LIN {X 0,Y 421.799,Z 977.518,A -85,B 0,C 180,E1 9515.942,E2 9515.942} C_VEL
LIN {X 0,Y 421.821,Z 978.492,A -85,B 0,C 180,E1 9519.003,E2 9519.003} C_VEL
LIN {X 0,Y 422.337,Z 975.375,A -85,B 0,C 180,E1 9522.556,E2 9522.556} C_VEL
LIN {X 0,Y 423.104,Z 967.595,A -85,B 0,C 180,E1 9526.055,E2 9526.055} C_VEL
LIN {X 0,Y 424.505,Z 953.17,A -85,B 0,C 180,E1 9529.758,E2 9529.758} C_VEL
LIN {X 0,Y 426.108,Z 934.517,A -85,B 0,C 180,E1 9532.847,E2 9532.847} C_VEL
LIN {X 0,Y 427.847,Z 910.65,A -85,B 0,C 180,E1 9535.461,E2 9535.461} C_VEL
LIN {X 0,Y 428.281,Z 890.231,A -85,B 0,C 180,E1 9537.014,E2 9537.014} C_VEL
LIN {X 0,Y 421.324,Z 861.271,A -85,B 0,C 180,E1 9538.781,E2 9538.781} C_VEL
LIN {X 0,Y 420.341,Z 857.28,A -85,B 0,C 180,E1 9538.956,E2 9538.956} C_VEL
LIN {X 0,Y 420.221,Z 857.28,A -85,B 0,C 180,E1 9544.157,E2 9544.157} C_VEL
LIN {X 0,Y 419.876,Z 857.28,A -85,B 0,C 180,E1 9550.41,E2 9550.41} C_VEL
LIN {X 0,Y 419.681,Z 857.28,A -85,B 0,C 180,E1 9556.795,E2 9556.795} C_VEL
LIN {X 0,Y 419.429,Z 857.28,A -85,B 0,C 180,E1 9563.414,E2 9563.414} C_VEL
LIN {X 0,Y 419.233,Z 857.28,A -85,B 0,C 180,E1 9570.388,E2 9570.388} C_VEL
LIN {X 0,Y 419.085,Z 857.28,A -85,B 0,C 180,E1 9577.363,E2 9577.363} C_VEL
LIN {X 0,Y 419.026,Z 857.28,A -85,B 0,C 180,E1 9583.726,E2 9583.726} C_VEL
LIN {X 0,Y 419.097,Z 857.28,A -85,B 0,C 180,E1 9589.438,E2 9589.438} C_VEL
LIN {X 0,Y 419.103,Z 857.28,A -85,B 0,C 180,E1 9596.203,E2 9596.203} C_VEL
LIN {X 0,Y 419.305,Z 857.723,A -85,B 0,C 180,E1 9598.793,E2 9598.793} C_VEL
LIN {X 0,Y 435.902,Z 903.66,A -85,B 0,C 180,E1 9600.619,E2 9600.619} C_VEL
LIN {X 0,Y 434.861,Z 940.44,A -85,B 0,C 180,E1 9601.516,E2 9601.516} C_VEL
LIN {X 0,Y 432.279,Z 973.093,A -85,B 0,C 180,E1 9603.034,E2 9603.034} C_VEL
LIN {X 0,Y 429.214,Z 1005.135,A -85,B 0,C 180,E1 9605.375,E2 9605.375} C_VEL
LIN {X 0,Y 428.851,Z 1008.694,A -85,B 0,C 180,E1 9605.694,E2 9605.694} C_VEL
LIN {X 0,Y 423.506,Z 1022.555,A -85,B 0,C 180,E1 9606.951,E2 9606.951} C_VEL
LIN {X 0,Y 418.257,Z 1035.44,A -85,B 0,C 180,E1 9608.402,E2 9608.402} C_VEL
LIN {X 0,Y 415.552,Z 1060.439,A -85,B 0,C 180,E1 9612.286,E2 9612.286} C_VEL
LIN {X 0,Y 414.019,Z 1079.134,A -85,B 0,C 180,E1 9616.393,E2 9616.393} C_VEL
LIN {X 0,Y 413.338,Z 1093.536,A -85,B 0,C 180,E1 9621.098,E2 9621.098} C_VEL
LIN {X 0,Y 413.202,Z 1101.646,A -85,B 0,C 180,E1 9625.798,E2 9625.798} C_VEL
LIN {X 0,Y 413.219,Z 1103.917,A -85,B 0,C 180,E1 9630.001,E2 9630.001} C_VEL
LIN {X 0,Y 413.204,Z 1101.557,A -85,B 0,C 180,E1 9634.203,E2 9634.203} C_VEL
LIN {X 0,Y 413.391,Z 1093.361,A -85,B 0,C 180,E1 9638.902,E2 9638.902} C_VEL
LIN {X 0,Y 414.016,Z 1078.868,A -85,B 0,C 180,E1 9643.605,E2 9643.605} C_VEL
LIN {X 0,Y 415.715,Z 1058.786,A -85,B 0,C 180,E1 9647.961,E2 9647.961} C_VEL
LIN {X 0,Y 418.387,Z 1034.343,A -85,B 0,C 180,E1 9651.712,E2 9651.712} C_VEL
LIN {X 0,Y 421.663,Z 1004.833,A -85,B 0,C 180,E1 9654.956,E2 9654.956} C_VEL
LIN {X 0,Y 425.056,Z 972.788,A -85,B 0,C 180,E1 9657.388,E2 9657.388} C_VEL
LIN {X 0,Y 427.787,Z 939.248,A -85,B 0,C 180,E1 9659.006,E2 9659.006} C_VEL
LIN {X 0,Y 428.561,Z 904.937,A -85,B 0,C 180,E1 9659.915,E2 9659.915} C_VEL
LIN {X 0,Y 412.812,Z 861.837,A -85,B 0,C 180,E1 9661.896,E2 9661.896} C_VEL
LIN {X 0,Y 411.31,Z 857.28,A -85,B 0,C 180,E1 9662.139,E2 9662.139} C_VEL
LIN {X 0,Y 411.036,Z 857.28,A -85,B 0,C 180,E1 9669.314,E2 9669.314} C_VEL
LIN {X 0,Y 411.046,Z 857.28,A -85,B 0,C 180,E1 9675.571,E2 9675.571} C_VEL
LIN {X 0,Y 411.109,Z 857.28,A -85,B 0,C 180,E1 9681.223,E2 9681.223} C_VEL
LIN {X 0,Y 411.195,Z 857.28,A -85,B 0,C 180,E1 9687.877,E2 9687.877} C_VEL
LIN {X 0,Y 411.371,Z 857.28,A -85,B 0,C 180,E1 9693.772,E2 9693.772} C_VEL
LIN {X 0,Y 411.659,Z 857.28,A -85,B 0,C 180,E1 9700.65,E2 9700.65} C_VEL
LIN {X 0,Y 411.735,Z 857.28,A -85,B 0,C 180,E1 9707.231,E2 9707.231} C_VEL
LIN {X 0,Y 412.172,Z 857.28,A -85,B 0,C 180,E1 9713.649,E2 9713.649} C_VEL
LIN {X 0,Y 412.461,Z 857.28,A -85,B 0,C 180,E1 9719.973,E2 9719.973} C_VEL
LIN {X 0,Y 412.137,Z 857.28,A -85,B 0,C 180,E1 9726.298,E2 9726.298} C_VEL
LIN {X 0,Y 411.881,Z 857.28,A -85,B 0,C 180,E1 9732.709,E2 9732.709} C_VEL
LIN {X 0,Y 411.647,Z 857.28,A -85,B 0,C 180,E1 9739.294,E2 9739.294} C_VEL
LIN {X 0,Y 411.376,Z 857.28,A -85,B 0,C 180,E1 9746.168,E2 9746.168} C_VEL
LIN {X 0,Y 411.191,Z 857.28,A -85,B 0,C 180,E1 9753.478,E2 9753.478} C_VEL
LIN {X 0,Y 411.021,Z 857.28,A -85,B 0,C 180,E1 9759.323,E2 9759.323} C_VEL
LIN {X 0,Y 411.073,Z 857.28,A -85,B 0,C 180,E1 9765.587,E2 9765.587} C_VEL
LIN {X 0,Y 411.258,Z 858.026,A -85,B 0,C 180,E1 9769.388,E2 9769.388} C_VEL
LIN {X 0,Y 420.757,Z 885.763,A -85,B 0,C 180,E1 9771.654,E2 9771.654} C_VEL
LIN {X 0,Y 423.982,Z 903.449,A -85,B 0,C 180,E1 9773.33,E2 9773.33} C_VEL
LIN {X 0,Y 421.34,Z 927.161,A -85,B 0,C 180,E1 9775.806,E2 9775.806} C_VEL
LIN {X 0,Y 418.651,Z 947.375,A -85,B 0,C 180,E1 9778.907,E2 9778.907} C_VEL
LIN {X 0,Y 416.418,Z 963.462,A -85,B 0,C 180,E1 9782.618,E2 9782.618} C_VEL
LIN {X 0,Y 415.038,Z 973.478,A -85,B 0,C 180,E1 9786.341,E2 9786.341} C_VEL
LIN {X 0,Y 414.274,Z 978.346,A -85,B 0,C 180,E1 9789.683,E2 9789.683} C_VEL
LIN {X 0,Y 413.931,Z 979.64,A -85,B 0,C 180,E1 9792.984,E2 9792.984} C_VEL
LIN {X 0,Y 414.318,Z 976.181,A -85,B 0,C 180,E1 9797.333,E2 9797.333} C_VEL
LIN {X 0,Y 415.259,Z 967.92,A -85,B 0,C 180,E1 9801.182,E2 9801.182} C_VEL
LIN {X 0,Y 416.858,Z 953.381,A -85,B 0,C 180,E1 9805.118,E2 9805.118} C_VEL
LIN {X 0,Y 419.039,Z 934.423,A -85,B 0,C 180,E1 9808.446,E2 9808.446} C_VEL
LIN {X 0,Y 421.351,Z 911.694,A -85,B 0,C 180,E1 9811.157,E2 9811.157} C_VEL
LIN {X 0,Y 422.02,Z 896.901,A -85,B 0,C 180,E1 9812.479,E2 9812.479} C_VEL
LIN {X 0,Y 415.522,Z 868.738,A -85,B 0,C 180,E1 9814.702,E2 9814.702} C_VEL
LIN {X 0,Y 412.172,Z 857.28,A -85,B 0,C 180,E1 9815.467,E2 9815.467} C_VEL
LIN {X 0,Y 411.961,Z 857.28,A -85,B 0,C 180,E1 9820.588,E2 9820.588} C_VEL
LIN {X 0,Y 411.718,Z 857.28,A -85,B 0,C 180,E1 9827.204,E2 9827.204} C_VEL
LIN {X 0,Y 411.416,Z 857.28,A -85,B 0,C 180,E1 9833.879,E2 9833.879} C_VEL
LIN {X 0,Y 411.283,Z 857.28,A -85,B 0,C 180,E1 9838.592,E2 9838.592} C_VEL
LIN {X 0,Y 411.132,Z 857.28,A -85,B 0,C 180,E1 9845.965,E2 9845.965} C_VEL
LIN {X 0,Y 411.032,Z 857.28,A -85,B 0,C 180,E1 9852.614,E2 9852.614} C_VEL
LIN {X 0,Y 411.302,Z 857.817,A -85,B 0,C 180,E1 9857,E2 9857} C_VEL
LIN {X 0,Y 418.345,Z 886.44,A -85,B 0,C 180,E1 9858.675,E2 9858.675} C_VEL
LIN {X 0,Y 419.854,Z 900.249,A -85,B 0,C 180,E1 9859.729,E2 9859.729} C_VEL
LIN {X 0,Y 418.125,Z 925.773,A -85,B 0,C 180,E1 9862.184,E2 9862.184} C_VEL
LIN {X 0,Y 416.519,Z 946.375,A -85,B 0,C 180,E1 9865.146,E2 9865.146} C_VEL
LIN {X 0,Y 415.31,Z 962.435,A -85,B 0,C 180,E1 9868.598,E2 9868.598} C_VEL
LIN {X 0,Y 414.455,Z 973.607,A -85,B 0,C 180,E1 9872.458,E2 9872.458} C_VEL
LIN {X 0,Y 413.982,Z 979.017,A -85,B 0,C 180,E1 9876.318,E2 9876.318} C_VEL
LIN {X 0,Y 413.979,Z 979.761,A -85,B 0,C 180,E1 9878.586,E2 9878.586} C_VEL
LIN {X 0,Y 414.406,Z 977.789,A -85,B 0,C 180,E1 9881.791,E2 9881.791} C_VEL
LIN {X 0,Y 415.312,Z 970.04,A -85,B 0,C 180,E1 9885.788,E2 9885.788} C_VEL
LIN {X 0,Y 416.722,Z 956.488,A -85,B 0,C 180,E1 9889.565,E2 9889.565} C_VEL
LIN {X 0,Y 418.38,Z 938.471,A -85,B 0,C 180,E1 9892.753,E2 9892.753} C_VEL
LIN {X 0,Y 420.149,Z 916.25,A -85,B 0,C 180,E1 9895.392,E2 9895.392} C_VEL
LIN {X 0,Y 420.82,Z 891.257,A -85,B 0,C 180,E1 9897.396,E2 9897.396} C_VEL
LIN {X 0,Y 413.932,Z 863.039,A -85,B 0,C 180,E1 9899.176,E2 9899.176} C_VEL
LIN {X 0,Y 412.429,Z 857.28,A -85,B 0,C 180,E1 9899.501,E2 9899.501} C_VEL
LIN {X 0,Y 412.121,Z 857.28,A -85,B 0,C 180,E1 9906.352,E2 9906.352} C_VEL
LIN {X 0,Y 411.856,Z 857.28,A -85,B 0,C 180,E1 9912.765,E2 9912.765} C_VEL
LIN {X 0,Y 411.654,Z 857.28,A -85,B 0,C 180,E1 9919.351,E2 9919.351} C_VEL
LIN {X 0,Y 411.368,Z 857.28,A -85,B 0,C 180,E1 9926.228,E2 9926.228} C_VEL
LIN {X 0,Y 411.217,Z 857.28,A -85,B 0,C 180,E1 9933.54,E2 9933.54} C_VEL
LIN {X 0,Y 411.052,Z 857.28,A -85,B 0,C 180,E1 9939.33,E2 9939.33} C_VEL
LIN {X 0,Y 411.092,Z 857.28,A -85,B 0,C 180,E1 9945.592,E2 9945.592} C_VEL
LIN {X 0,Y 411.112,Z 857.28,A -85,B 0,C 180,E1 9951.239,E2 9951.239} C_VEL
LIN {X 0,Y 411.368,Z 857.28,A -85,B 0,C 180,E1 9958.268,E2 9958.268} C_VEL
LIN {X 0,Y 428.788,Z 907.527,A -85,B 0,C 180,E1 9960.271,E2 9960.271} C_VEL
LIN {X 0,Y 427.327,Z 943.567,A -85,B 0,C 180,E1 9961.236,E2 9961.236} C_VEL
LIN {X 0,Y 424.531,Z 976.772,A -85,B 0,C 180,E1 9962.901,E2 9962.901} C_VEL
LIN {X 0,Y 421.193,Z 1009.104,A -85,B 0,C 180,E1 9965.441,E2 9965.441} C_VEL
LIN {X 0,Y 418.257,Z 1035.44,A -85,B 0,C 180,E1 9968.402,E2 9968.402} C_VEL
LIN {X 0,Y 416.387,Z 1041.625,A -85,B 0,C 180,E1 9969.217,E2 9969.217} C_VEL
LIN {X 0,Y 408.17,Z 1056.964,A -85,B 0,C 180,E1 9971.556,E2 9971.556} C_VEL
LIN {X 0,Y 407.937,Z 1058.282,A -85,B 0,C 180,E1 9971.801,E2 9971.801} C_VEL
LIN {X 0,Y 406.3,Z 1076.772,A -85,B 0,C 180,E1 9975.845,E2 9975.845} C_VEL
LIN {X 0,Y 405.5,Z 1090.903,A -85,B 0,C 180,E1 9980.328,E2 9980.328} C_VEL
LIN {X 0,Y 405.399,Z 1099.167,A -85,B 0,C 180,E1 9984.643,E2 9984.643} C_VEL
LIN {X 0,Y 405.33,Z 1102.132,A -85,B 0,C 180,E1 9987.86,E2 9987.86} C_VEL
LIN {X 0,Y 405.334,Z 1102.085,A -85,B 0,C 180,E1 9992.141,E2 9992.141} C_VEL
LIN {X 0,Y 405.37,Z 1097.398,A -85,B 0,C 180,E1 9996.434,E2 9996.434} C_VEL
LIN {X 0,Y 405.594,Z 1087.82,A -85,B 0,C 180,E1 10000.758,E2 10000.758} C_VEL
LIN {X 0,Y 406.651,Z 1071.54,A -85,B 0,C 180,E1 10005.385,E2 10005.385} C_VEL
LIN {X 0,Y 408.664,Z 1050.837,A -85,B 0,C 180,E1 10009.479,E2 10009.479} C_VEL
LIN {X 0,Y 411.694,Z 1025.006,A -85,B 0,C 180,E1 10013.148,E2 10013.148} C_VEL
LIN {X 0,Y 415.216,Z 995.793,A -85,B 0,C 180,E1 10016.108,E2 10016.108} C_VEL
LIN {X 0,Y 418.709,Z 963.598,A -85,B 0,C 180,E1 10018.343,E2 10018.343} C_VEL
LIN {X 0,Y 421.277,Z 930.208,A -85,B 0,C 180,E1 10019.771,E2 10019.771} C_VEL
LIN {X 0,Y 421.345,Z 906.279,A -85,B 0,C 180,E1 10020.4,E2 10020.4} C_VEL
LIN {X 0,Y 407.006,Z 866.784,A -85,B 0,C 180,E1 10022.269,E2 10022.269} C_VEL
LIN {X 0,Y 403.353,Z 857.28,A -85,B 0,C 180,E1 10022.88,E2 10022.88} C_VEL
LIN {X 0,Y 403.089,Z 857.28,A -85,B 0,C 180,E1 10029.685,E2 10029.685} C_VEL
LIN {X 0,Y 403.143,Z 857.28,A -85,B 0,C 180,E1 10035.528,E2 10035.528} C_VEL
LIN {X 0,Y 403.133,Z 857.28,A -85,B 0,C 180,E1 10042.067,E2 10042.067} C_VEL
LIN {X 0,Y 403.303,Z 857.28,A -85,B 0,C 180,E1 10048.275,E2 10048.275} C_VEL
LIN {X 0,Y 403.503,Z 857.28,A -85,B 0,C 180,E1 10055.603,E2 10055.603} C_VEL
LIN {X 0,Y 403.726,Z 857.28,A -85,B 0,C 180,E1 10062.52,E2 10062.52} C_VEL
LIN {X 0,Y 403.89,Z 857.28,A -85,B 0,C 180,E1 10069.174,E2 10069.174} C_VEL
LIN {X 0,Y 404.284,Z 857.28,A -85,B 0,C 180,E1 10075.679,E2 10075.679} C_VEL
LIN {X 0,Y 404.458,Z 857.28,A -85,B 0,C 180,E1 10082.117,E2 10082.117} C_VEL
LIN {X 0,Y 404.116,Z 857.28,A -85,B 0,C 180,E1 10088.588,E2 10088.588} C_VEL
LIN {X 0,Y 403.867,Z 857.28,A -85,B 0,C 180,E1 10095.179,E2 10095.179} C_VEL
LIN {X 0,Y 403.608,Z 857.28,A -85,B 0,C 180,E1 10101.993,E2 10101.993} C_VEL
LIN {X 0,Y 403.322,Z 857.28,A -85,B 0,C 180,E1 10109.165,E2 10109.165} C_VEL
LIN {X 0,Y 403.218,Z 857.28,A -85,B 0,C 180,E1 10114.299,E2 10114.299} C_VEL
LIN {X 0,Y 403.087,Z 857.28,A -85,B 0,C 180,E1 10121.301,E2 10121.301} C_VEL
LIN {X 0,Y 403.18,Z 857.28,A -85,B 0,C 180,E1 10127.47,E2 10127.47} C_VEL
LIN {X 0,Y 403.25,Z 857.838,A -85,B 0,C 180,E1 10128.673,E2 10128.673} C_VEL
LIN {X 0,Y 412.99,Z 885.391,A -85,B 0,C 180,E1 10130.993,E2 10130.993} C_VEL
LIN {X 0,Y 416.797,Z 905.603,A -85,B 0,C 180,E1 10132.975,E2 10132.975} C_VEL
LIN {X 0,Y 413.764,Z 930.558,A -85,B 0,C 180,E1 10135.701,E2 10135.701} C_VEL
LIN {X 0,Y 410.953,Z 950.524,A -85,B 0,C 180,E1 10138.948,E2 10138.948} C_VEL
LIN {X 0,Y 408.665,Z 965.697,A -85,B 0,C 180,E1 10142.663,E2 10142.663} C_VEL
LIN {X 0,Y 407.065,Z 976.221,A -85,B 0,C 180,E1 10147.011,E2 10147.011} C_VEL
LIN {X 0,Y 406.352,Z 980.147,A -85,B 0,C 180,E1 10150.406,E2 10150.406} C_VEL
LIN {X 0,Y 406.187,Z 980.065,A -85,B 0,C 180,E1 10154.874,E2 10154.874} C_VEL
LIN {X 0,Y 406.935,Z 974.024,A -85,B 0,C 180,E1 10159.278,E2 10159.278} C_VEL
LIN {X 0,Y 408.182,Z 963.556,A -85,B 0,C 180,E1 10163.075,E2 10163.075} C_VEL
LIN {X 0,Y 410.029,Z 946.849,A -85,B 0,C 180,E1 10166.87,E2 10166.87} C_VEL
LIN {X 0,Y 412.625,Z 925.085,A -85,B 0,C 180,E1 10170.131,E2 10170.131} C_VEL
LIN {X 0,Y 414.937,Z 900.466,A -85,B 0,C 180,E1 10172.614,E2 10172.614} C_VEL
LIN {X 0,Y 408.725,Z 872.434,A -85,B 0,C 180,E1 10174.946,E2 10174.946} C_VEL
LIN {X 0,Y 404.281,Z 857.28,A -85,B 0,C 180,E1 10176.045,E2 10176.045} C_VEL
LIN {X 0,Y 403.946,Z 857.28,A -85,B 0,C 180,E1 10183.186,E2 10183.186} C_VEL
LIN {X 0,Y 403.666,Z 857.28,A -85,B 0,C 180,E1 10189.728,E2 10189.728} C_VEL
LIN {X 0,Y 403.392,Z 857.28,A -85,B 0,C 180,E1 10196.769,E2 10196.769} C_VEL
LIN {X 0,Y 403.237,Z 857.28,A -85,B 0,C 180,E1 10201.713,E2 10201.713} C_VEL
LIN {X 0,Y 403.069,Z 857.28,A -85,B 0,C 180,E1 10208,E2 10208} C_VEL
LIN {X 0,Y 403.179,Z 857.28,A -85,B 0,C 180,E1 10214.543,E2 10214.543} C_VEL
LIN {X 0,Y 403.347,Z 857.28,A -85,B 0,C 180,E1 10216.554,E2 10216.554} C_VEL
LIN {X 0,Y 410.553,Z 886.738,A -85,B 0,C 180,E1 10218.313,E2 10218.313} C_VEL
LIN {X 0,Y 412.256,Z 902.112,A -85,B 0,C 180,E1 10219.511,E2 10219.511} C_VEL
LIN {X 0,Y 410.519,Z 926.722,A -85,B 0,C 180,E1 10221.928,E2 10221.928} C_VEL
LIN {X 0,Y 408.827,Z 947.408,A -85,B 0,C 180,E1 10224.943,E2 10224.943} C_VEL
LIN {X 0,Y 407.561,Z 963.335,A -85,B 0,C 180,E1 10228.403,E2 10228.403} C_VEL
LIN {X 0,Y 406.687,Z 974.589,A -85,B 0,C 180,E1 10232.311,E2 10232.311} C_VEL
LIN {X 0,Y 406.202,Z 979.817,A -85,B 0,C 180,E1 10235.835,E2 10235.835} C_VEL
LIN {X 0,Y 406.194,Z 980.973,A -85,B 0,C 180,E1 10238.726,E2 10238.726} C_VEL
LIN {X 0,Y 406.813,Z 977.958,A -85,B 0,C 180,E1 10242.714,E2 10242.714} C_VEL
LIN {X 0,Y 407.768,Z 969.392,A -85,B 0,C 180,E1 10246.652,E2 10246.652} C_VEL
LIN {X 0,Y 409.425,Z 954.746,A -85,B 0,C 180,E1 10250.452,E2 10250.452} C_VEL
LIN {X 0,Y 411.31,Z 935.202,A -85,B 0,C 180,E1 10253.69,E2 10253.69} C_VEL
LIN {X 0,Y 413.177,Z 912.352,A -85,B 0,C 180,E1 10256.22,E2 10256.22} C_VEL
LIN {X 0,Y 413.681,Z 893.995,A -85,B 0,C 180,E1 10257.668,E2 10257.668} C_VEL
LIN {X 0,Y 407.079,Z 866.072,A -85,B 0,C 180,E1 10259.518,E2 10259.518} C_VEL
LIN {X 0,Y 404.546,Z 857.28,A -85,B 0,C 180,E1 10260.027,E2 10260.027} C_VEL
LIN {X 0,Y 404.205,Z 857.28,A -85,B 0,C 180,E1 10266.477,E2 10266.477} C_VEL
LIN {X 0,Y 403.943,Z 857.28,A -85,B 0,C 180,E1 10273.019,E2 10273.019} C_VEL
LIN {X 0,Y 403.691,Z 857.28,A -85,B 0,C 180,E1 10279.748,E2 10279.748} C_VEL
LIN {X 0,Y 403.436,Z 857.28,A -85,B 0,C 180,E1 10286.785,E2 10286.785} C_VEL
LIN {X 0,Y 403.305,Z 857.28,A -85,B 0,C 180,E1 10291.725,E2 10291.725} C_VEL
LIN {X 0,Y 403.088,Z 857.28,A -85,B 0,C 180,E1 10297.928,E2 10297.928} C_VEL
LIN {X 0,Y 403.176,Z 857.28,A -85,B 0,C 180,E1 10304.479,E2 10304.479} C_VEL
LIN {X 0,Y 403.172,Z 857.28,A -85,B 0,C 180,E1 10310.327,E2 10310.327} C_VEL
LIN {X 0,Y 403.41,Z 857.488,A -85,B 0,C 180,E1 10317.744,E2 10317.744} C_VEL
LIN {X 0,Y 421.549,Z 909.75,A -85,B 0,C 180,E1 10319.877,E2 10319.877} C_VEL
LIN {X 0,Y 419.914,Z 945.02,A -85,B 0,C 180,E1 10320.888,E2 10320.888} C_VEL
LIN {X 0,Y 416.875,Z 978.864,A -85,B 0,C 180,E1 10322.687,E2 10322.687} C_VEL
LIN {X 0,Y 413.474,Z 1009.986,A -85,B 0,C 180,E1 10325.24,E2 10325.24} C_VEL
LIN {X 0,Y 410.12,Z 1038.585,A -85,B 0,C 180,E1 10328.62,E2 10328.62} C_VEL
LIN {X 0,Y 407.937,Z 1058.282,A -85,B 0,C 180,E1 10331.801,E2 10331.801} C_VEL
LIN {X 0,Y 403.019,Z 1068.016,A -85,B 0,C 180,E1 10333.752,E2 10333.752} C_VEL
LIN {X 0,Y 398.406,Z 1076.498,A -85,B 0,C 180,E1 10335.847,E2 10335.847} C_VEL
LIN {X 0,Y 397.627,Z 1090.953,A -85,B 0,C 180,E1 10340.688,E2 10340.688} C_VEL
LIN {X 0,Y 397.57,Z 1097.979,A -85,B 0,C 180,E1 10344.537,E2 10344.537} C_VEL
LIN {X 0,Y 397.506,Z 1100.956,A -85,B 0,C 180,E1 10347.818,E2 10347.818} C_VEL
LIN {X 0,Y 397.51,Z 1100.908,A -85,B 0,C 180,E1 10352.184,E2 10352.184} C_VEL
LIN {X 0,Y 397.55,Z 1096.206,A -85,B 0,C 180,E1 10356.561,E2 10356.561} C_VEL
LIN {X 0,Y 397.751,Z 1086.607,A -85,B 0,C 180,E1 10360.973,E2 10360.973} C_VEL
LIN {X 0,Y 398.894,Z 1070.287,A -85,B 0,C 180,E1 10365.691,E2 10365.691} C_VEL
LIN {X 0,Y 401.197,Z 1047.885,A -85,B 0,C 180,E1 10370.144,E2 10370.144} C_VEL
LIN {X 0,Y 404.421,Z 1022.323,A -85,B 0,C 180,E1 10373.772,E2 10373.772} C_VEL
LIN {X 0,Y 408.187,Z 992.517,A -85,B 0,C 180,E1 10376.773,E2 10376.773} C_VEL
LIN {X 0,Y 411.785,Z 960.401,A -85,B 0,C 180,E1 10378.967,E2 10378.967} C_VEL
LIN {X 0,Y 414.481,Z 926.066,A -85,B 0,C 180,E1 10380.394,E2 10380.394} C_VEL
LIN {X 0,Y 414.518,Z 908.545,A -85,B 0,C 180,E1 10380.854,E2 10380.854} C_VEL
LIN {X 0,Y 400.695,Z 870.24,A -85,B 0,C 180,E1 10382.732,E2 10382.732} C_VEL
LIN {X 0,Y 395.38,Z 857.28,A -85,B 0,C 180,E1 10383.539,E2 10383.539} C_VEL
LIN {X 0,Y 395.178,Z 857.28,A -85,B 0,C 180,E1 10390.643,E2 10390.643} C_VEL
LIN {X 0,Y 395.204,Z 857.28,A -85,B 0,C 180,E1 10396.713,E2 10396.713} C_VEL
LIN {X 0,Y 395.224,Z 857.28,A -85,B 0,C 180,E1 10403.563,E2 10403.563} C_VEL
LIN {X 0,Y 395.422,Z 857.28,A -85,B 0,C 180,E1 10410.129,E2 10410.129} C_VEL
LIN {X 0,Y 395.654,Z 857.28,A -85,B 0,C 180,E1 10417.48,E2 10417.48} C_VEL
LIN {X 0,Y 395.796,Z 857.28,A -85,B 0,C 180,E1 10424.446,E2 10424.446} C_VEL
LIN {X 0,Y 396.18,Z 857.28,A -85,B 0,C 180,E1 10431.182,E2 10431.182} C_VEL
LIN {X 0,Y 396.624,Z 857.28,A -85,B 0,C 180,E1 10437.785,E2 10437.785} C_VEL
LIN {X 0,Y 396.46,Z 857.28,A -85,B 0,C 180,E1 10444.351,E2 10444.351} C_VEL
LIN {X 0,Y 396.105,Z 857.28,A -85,B 0,C 180,E1 10450.985,E2 10450.985} C_VEL
LIN {X 0,Y 395.861,Z 857.28,A -85,B 0,C 180,E1 10457.78,E2 10457.78} C_VEL
LIN {X 0,Y 395.562,Z 857.28,A -85,B 0,C 180,E1 10464.858,E2 10464.858} C_VEL
LIN {X 0,Y 395.39,Z 857.28,A -85,B 0,C 180,E1 10469.809,E2 10469.809} C_VEL
LIN {X 0,Y 395.164,Z 857.28,A -85,B 0,C 180,E1 10476.425,E2 10476.425} C_VEL
LIN {X 0,Y 395.176,Z 857.28,A -85,B 0,C 180,E1 10483.54,E2 10483.54} C_VEL
LIN {X 0,Y 395.303,Z 857.752,A -85,B 0,C 180,E1 10487.932,E2 10487.932} C_VEL
LIN {X 0,Y 405.656,Z 886.594,A -85,B 0,C 180,E1 10490.452,E2 10490.452} C_VEL
LIN {X 0,Y 409.752,Z 906.655,A -85,B 0,C 180,E1 10492.504,E2 10492.504} C_VEL
LIN {X 0,Y 406.609,Z 931.138,A -85,B 0,C 180,E1 10495.212,E2 10495.212} C_VEL
LIN {X 0,Y 403.574,Z 951.34,A -85,B 0,C 180,E1 10498.533,E2 10498.533} C_VEL
LIN {X 0,Y 400.976,Z 967.421,A -85,B 0,C 180,E1 10502.576,E2 10502.576} C_VEL
LIN {X 0,Y 399.409,Z 976.939,A -85,B 0,C 180,E1 10506.544,E2 10506.544} C_VEL
LIN {X 0,Y 398.598,Z 981.128,A -85,B 0,C 180,E1 10510.009,E2 10510.009} C_VEL
LIN {X 0,Y 398.358,Z 981.404,A -85,B 0,C 180,E1 10514.569,E2 10514.569} C_VEL
LIN {X 0,Y 399.089,Z 975.816,A -85,B 0,C 180,E1 10519.064,E2 10519.064} C_VEL
LIN {X 0,Y 400.311,Z 965.763,A -85,B 0,C 180,E1 10522.938,E2 10522.938} C_VEL
LIN {X 0,Y 402.252,Z 949.494,A -85,B 0,C 180,E1 10526.832,E2 10526.832} C_VEL
LIN {X 0,Y 404.884,Z 928.588,A -85,B 0,C 180,E1 10530.133,E2 10530.133} C_VEL
LIN {X 0,Y 407.504,Z 903.528,A -85,B 0,C 180,E1 10532.801,E2 10532.801} C_VEL
LIN {X 0,Y 402.018,Z 876.594,A -85,B 0,C 180,E1 10535.158,E2 10535.158} C_VEL
LIN {X 0,Y 396.318,Z 857.28,A -85,B 0,C 180,E1 10536.58,E2 10536.58} C_VEL
LIN {X 0,Y 396.051,Z 857.28,A -85,B 0,C 180,E1 10543.26,E2 10543.26} C_VEL
LIN {X 0,Y 395.729,Z 857.28,A -85,B 0,C 180,E1 10550.141,E2 10550.141} C_VEL
LIN {X 0,Y 395.4,Z 857.28,A -85,B 0,C 180,E1 10557.355,E2 10557.355} C_VEL
LIN {X 0,Y 395.235,Z 857.28,A -85,B 0,C 180,E1 10562.656,E2 10562.656} C_VEL
LIN {X 0,Y 395.162,Z 857.28,A -85,B 0,C 180,E1 10570.05,E2 10570.05} C_VEL
LIN {X 0,Y 395.421,Z 857.731,A -85,B 0,C 180,E1 10576.204,E2 10576.204} C_VEL
LIN {X 0,Y 402.625,Z 886.578,A -85,B 0,C 180,E1 10577.908,E2 10577.908} C_VEL
LIN {X 0,Y 404.763,Z 902.529,A -85,B 0,C 180,E1 10579.168,E2 10579.168} C_VEL
LIN {X 0,Y 402.857,Z 928.419,A -85,B 0,C 180,E1 10581.752,E2 10581.752} C_VEL
LIN {X 0,Y 401.051,Z 949.418,A -85,B 0,C 180,E1 10584.913,E2 10584.913} C_VEL
LIN {X 0,Y 399.733,Z 966.013,A -85,B 0,C 180,E1 10588.695,E2 10588.695} C_VEL
LIN {X 0,Y 398.864,Z 976.061,A -85,B 0,C 180,E1 10592.39,E2 10592.39} C_VEL
LIN {X 0,Y 398.408,Z 980.97,A -85,B 0,C 180,E1 10595.792,E2 10595.792} C_VEL
LIN {X 0,Y 398.56,Z 981.853,A -85,B 0,C 180,E1 10600.046,E2 10600.046} C_VEL
LIN {X 0,Y 399.323,Z 977.179,A -85,B 0,C 180,E1 10604.08,E2 10604.08} C_VEL
LIN {X 0,Y 400.609,Z 966.545,A -85,B 0,C 180,E1 10608.147,E2 10608.147} C_VEL
LIN {X 0,Y 402.291,Z 951.37,A -85,B 0,C 180,E1 10611.646,E2 10611.646} C_VEL
LIN {X 0,Y 404.458,Z 930.239,A -85,B 0,C 180,E1 10614.829,E2 10614.829} C_VEL
LIN {X 0,Y 406.406,Z 906.173,A -85,B 0,C 180,E1 10617.226,E2 10617.226} C_VEL
LIN {X 0,Y 405.655,Z 891.937,A -85,B 0,C 180,E1 10618.333,E2 10618.333} C_VEL
LIN {X 0,Y 398.867,Z 864.613,A -85,B 0,C 180,E1 10620.13,E2 10620.13} C_VEL
LIN {X 0,Y 396.573,Z 857.28,A -85,B 0,C 180,E1 10620.575,E2 10620.575} C_VEL
LIN {X 0,Y 396.287,Z 857.28,A -85,B 0,C 180,E1 10626.607,E2 10626.607} C_VEL
LIN {X 0,Y 395.999,Z 857.28,A -85,B 0,C 180,E1 10633.285,E2 10633.285} C_VEL
LIN {X 0,Y 395.774,Z 857.28,A -85,B 0,C 180,E1 10640.16,E2 10640.16} C_VEL
LIN {X 0,Y 395.448,Z 857.28,A -85,B 0,C 180,E1 10647.37,E2 10647.37} C_VEL
LIN {X 0,Y 395.326,Z 857.28,A -85,B 0,C 180,E1 10652.587,E2 10652.587} C_VEL
LIN {X 0,Y 395.213,Z 857.28,A -85,B 0,C 180,E1 10659.987,E2 10659.987} C_VEL
LIN {X 0,Y 395.24,Z 857.28,A -85,B 0,C 180,E1 10666.721,E2 10666.721} C_VEL
LIN {X 0,Y 395.23,Z 857.28,A -85,B 0,C 180,E1 10673.574,E2 10673.574} C_VEL
LIN {X 0,Y 395.451,Z 857.28,A -85,B 0,C 180,E1 10677.177,E2 10677.177} C_VEL
LIN {X 0,Y 414.296,Z 909.828,A -85,B 0,C 180,E1 10679.434,E2 10679.434} C_VEL
LIN {X 0,Y 412.562,Z 945.735,A -85,B 0,C 180,E1 10680.501,E2 10680.501} C_VEL
LIN {X 0,Y 409.54,Z 977.826,A -85,B 0,C 180,E1 10682.251,E2 10682.251} C_VEL
LIN {X 0,Y 405.943,Z 1009.456,A -85,B 0,C 180,E1 10684.897,E2 10684.897} C_VEL
LIN {X 0,Y 402.556,Z 1036.966,A -85,B 0,C 180,E1 10688.198,E2 10688.198} C_VEL
LIN {X 0,Y 399.912,Z 1059.738,A -85,B 0,C 180,E1 10692.003,E2 10692.003} C_VEL
LIN {X 0,Y 398.406,Z 1076.498,A -85,B 0,C 180,E1 10695.847,E2 10695.847} C_VEL
LIN {X 0,Y 395.545,Z 1082.115,A -85,B 0,C 180,E1 10697.513,E2 10697.513} C_VEL
LIN {X 0,Y 389.884,Z 1088.855,A -85,B 0,C 180,E1 10700.117,E2 10700.117} C_VEL
LIN {X 0,Y 389.777,Z 1089.526,A -85,B 0,C 180,E1 10700.423,E2 10700.423} C_VEL
LIN {X 0,Y 389.742,Z 1096.776,A -85,B 0,C 180,E1 10704.427,E2 10704.427} C_VEL
LIN {X 0,Y 389.696,Z 1099.774,A -85,B 0,C 180,E1 10707.774,E2 10707.774} C_VEL
LIN {X 0,Y 389.7,Z 1099.736,A -85,B 0,C 180,E1 10712.227,E2 10712.227} C_VEL
LIN {X 0,Y 389.716,Z 1095.022,A -85,B 0,C 180,E1 10716.694,E2 10716.694} C_VEL
LIN {X 0,Y 389.908,Z 1085.395,A -85,B 0,C 180,E1 10721.196,E2 10721.196} C_VEL
LIN {X 0,Y 391.134,Z 1069.07,A -85,B 0,C 180,E1 10726.011,E2 10726.011} C_VEL
LIN {X 0,Y 393.354,Z 1048.307,A -85,B 0,C 180,E1 10730.27,E2 10730.27} C_VEL
LIN {X 0,Y 396.754,Z 1022.833,A -85,B 0,C 180,E1 10734.023,E2 10734.023} C_VEL
LIN {X 0,Y 400.75,Z 992.969,A -85,B 0,C 180,E1 10737.142,E2 10737.142} C_VEL
LIN {X 0,Y 404.541,Z 961.247,A -85,B 0,C 180,E1 10739.396,E2 10739.396} C_VEL
LIN {X 0,Y 407.347,Z 928.595,A -85,B 0,C 180,E1 10740.825,E2 10740.825} C_VEL
LIN {X 0,Y 407.443,Z 910.061,A -85,B 0,C 180,E1 10741.366,E2 10741.366} C_VEL
LIN {X 0,Y 394.116,Z 873.196,A -85,B 0,C 180,E1 10743.253,E2 10743.253} C_VEL
LIN {X 0,Y 387.397,Z 857.28,A -85,B 0,C 180,E1 10744.248,E2 10744.248} C_VEL
LIN {X 0,Y 387.178,Z 857.28,A -85,B 0,C 180,E1 10751.668,E2 10751.668} C_VEL
LIN {X 0,Y 387.228,Z 857.28,A -85,B 0,C 180,E1 10758.324,E2 10758.324} C_VEL
LIN {X 0,Y 387.359,Z 857.28,A -85,B 0,C 180,E1 10765.169,E2 10765.169} C_VEL
LIN {X 0,Y 387.541,Z 857.28,A -85,B 0,C 180,E1 10772.023,E2 10772.023} C_VEL
LIN {X 0,Y 387.835,Z 857.28,A -85,B 0,C 180,E1 10779.546,E2 10779.546} C_VEL
LIN {X 0,Y 387.914,Z 857.28,A -85,B 0,C 180,E1 10786.433,E2 10786.433} C_VEL
LIN {X 0,Y 388.451,Z 857.28,A -85,B 0,C 180,E1 10793.259,E2 10793.259} C_VEL
LIN {X 0,Y 388.763,Z 857.28,A -85,B 0,C 180,E1 10799.971,E2 10799.971} C_VEL
LIN {X 0,Y 388.404,Z 857.28,A -85,B 0,C 180,E1 10806.684,E2 10806.684} C_VEL
LIN {X 0,Y 388.072,Z 857.28,A -85,B 0,C 180,E1 10813.503,E2 10813.503} C_VEL
LIN {X 0,Y 387.797,Z 857.28,A -85,B 0,C 180,E1 10820.532,E2 10820.532} C_VEL
LIN {X 0,Y 387.523,Z 857.28,A -85,B 0,C 180,E1 10827.914,E2 10827.914} C_VEL
LIN {X 0,Y 387.275,Z 857.28,A -85,B 0,C 180,E1 10835.851,E2 10835.851} C_VEL
LIN {X 0,Y 387.154,Z 857.28,A -85,B 0,C 180,E1 10842.007,E2 10842.007} C_VEL
LIN {X 0,Y 387.348,Z 857.28,A -85,B 0,C 180,E1 10847.133,E2 10847.133} C_VEL
LIN {X 0,Y 398.064,Z 886.834,A -85,B 0,C 180,E1 10849.786,E2 10849.786} C_VEL
LIN {X 0,Y 402.64,Z 908.425,A -85,B 0,C 180,E1 10852.079,E2 10852.079} C_VEL
LIN {X 0,Y 399.36,Z 932.498,A -85,B 0,C 180,E1 10854.81,E2 10854.81} C_VEL
LIN {X 0,Y 396.245,Z 951.943,A -85,B 0,C 180,E1 10858.055,E2 10858.055} C_VEL
LIN {X 0,Y 393.647,Z 966.945,A -85,B 0,C 180,E1 10861.767,E2 10861.767} C_VEL
LIN {X 0,Y 391.781,Z 977.624,A -85,B 0,C 180,E1 10866.059,E2 10866.059} C_VEL
LIN {X 0,Y 390.883,Z 982.112,A -85,B 0,C 180,E1 10869.597,E2 10869.597} C_VEL
LIN {X 0,Y 390.517,Z 982.738,A -85,B 0,C 180,E1 10874.252,E2 10874.252} C_VEL
LIN {X 0,Y 391.21,Z 977.525,A -85,B 0,C 180,E1 10878.841,E2 10878.841} C_VEL
LIN {X 0,Y 392.46,Z 967.87,A -85,B 0,C 180,E1 10882.796,E2 10882.796} C_VEL
LIN {X 0,Y 394.399,Z 952.815,A -85,B 0,C 180,E1 10886.636,E2 10886.636} C_VEL
LIN {X 0,Y 396.975,Z 933.05,A -85,B 0,C 180,E1 10889.999,E2 10889.999} C_VEL
LIN {X 0,Y 399.784,Z 908.244,A -85,B 0,C 180,E1 10892.848,E2 10892.848} C_VEL
LIN {X 0,Y 398.444,Z 895.498,A -85,B 0,C 180,E1 10894.085,E2 10894.085} C_VEL
LIN {X 0,Y 391.725,Z 868.476,A -85,B 0,C 180,E1 10896.291,E2 10896.291} C_VEL
LIN {X 0,Y 388.372,Z 857.28,A -85,B 0,C 180,E1 10897.059,E2 10897.059} C_VEL
LIN {X 0,Y 388.116,Z 857.28,A -85,B 0,C 180,E1 10903.536,E2 10903.536} C_VEL
LIN {X 0,Y 387.758,Z 857.28,A -85,B 0,C 180,E1 10910.574,E2 10910.574} C_VEL
LIN {X 0,Y 387.463,Z 857.28,A -85,B 0,C 180,E1 10917.963,E2 10917.963} C_VEL
LIN {X 0,Y 387.268,Z 857.28,A -85,B 0,C 180,E1 10925.904,E2 10925.904} C_VEL
LIN {X 0,Y 387.175,Z 857.28,A -85,B 0,C 180,E1 10932.082,E2 10932.082} C_VEL
LIN {X 0,Y 387.446,Z 857.28,A -85,B 0,C 180,E1 10935.759,E2 10935.759} C_VEL
LIN {X 0,Y 394.762,Z 886.609,A -85,B 0,C 180,E1 10937.508,E2 10937.508} C_VEL
LIN {X 0,Y 397.189,Z 904.358,A -85,B 0,C 180,E1 10938.941,E2 10938.941} C_VEL
LIN {X 0,Y 395.259,Z 929.232,A -85,B 0,C 180,E1 10941.473,E2 10941.473} C_VEL
LIN {X 0,Y 393.347,Z 950.858,A -85,B 0,C 180,E1 10944.785,E2 10944.785} C_VEL
LIN {X 0,Y 391.954,Z 967.218,A -85,B 0,C 180,E1 10948.591,E2 10948.591} C_VEL
LIN {X 0,Y 391.069,Z 977.282,A -85,B 0,C 180,E1 10952.361,E2 10952.361} C_VEL
LIN {X 0,Y 390.683,Z 981.15,A -85,B 0,C 180,E1 10954.81,E2 10954.81} C_VEL
LIN {X 0,Y 390.601,Z 983.414,A -85,B 0,C 180,E1 10958.48,E2 10958.48} C_VEL
LIN {X 0,Y 391.343,Z 980.175,A -85,B 0,C 180,E1 10963.169,E2 10963.169} C_VEL
LIN {X 0,Y 392.504,Z 971.47,A -85,B 0,C 180,E1 10967.22,E2 10967.22} C_VEL
LIN {X 0,Y 394.265,Z 957.644,A -85,B 0,C 180,E1 10970.932,E2 10970.932} C_VEL
LIN {X 0,Y 396.395,Z 938.521,A -85,B 0,C 180,E1 10974.253,E2 10974.253} C_VEL
LIN {X 0,Y 398.524,Z 915.72,A -85,B 0,C 180,E1 10976.899,E2 10976.899} C_VEL
LIN {X 0,Y 398.916,Z 896.3,A -85,B 0,C 180,E1 10978.518,E2 10978.518} C_VEL
LIN {X 0,Y 392.324,Z 868.495,A -85,B 0,C 180,E1 10980.469,E2 10980.469} C_VEL
LIN {X 0,Y 388.639,Z 857.28,A -85,B 0,C 180,E1 10981.102,E2 10981.102} C_VEL
LIN {X 0,Y 388.364,Z 857.28,A -85,B 0,C 180,E1 10986.742,E2 10986.742} C_VEL
LIN {X 0,Y 388.072,Z 857.28,A -85,B 0,C 180,E1 10993.562,E2 10993.562} C_VEL
LIN {X 0,Y 387.799,Z 857.28,A -85,B 0,C 180,E1 11000.593,E2 11000.593} C_VEL
LIN {X 0,Y 387.543,Z 857.28,A -85,B 0,C 180,E1 11007.977,E2 11007.977} C_VEL
LIN {X 0,Y 387.345,Z 857.28,A -85,B 0,C 180,E1 11014.83,E2 11014.83} C_VEL
LIN {X 0,Y 387.199,Z 857.28,A -85,B 0,C 180,E1 11022.017,E2 11022.017} C_VEL
LIN {X 0,Y 387.251,Z 857.28,A -85,B 0,C 180,E1 11028.344,E2 11028.344} C_VEL
LIN {X 0,Y 387.363,Z 857.28,A -85,B 0,C 180,E1 11035.182,E2 11035.182} C_VEL
LIN {X 0,Y 387.514,Z 857.28,A -85,B 0,C 180,E1 11036.588,E2 11036.588} C_VEL
LIN {X 0,Y 406.922,Z 911.189,A -85,B 0,C 180,E1 11039,E2 11039} C_VEL
LIN {X 0,Y 405.258,Z 945.909,A -85,B 0,C 180,E1 11040.091,E2 11040.091} C_VEL
LIN {X 0,Y 401.96,Z 979.058,A -85,B 0,C 180,E1 11041.965,E2 11041.965} C_VEL
LIN {X 0,Y 398.217,Z 1010.217,A -85,B 0,C 180,E1 11044.677,E2 11044.677} C_VEL
LIN {X 0,Y 394.739,Z 1037.271,A -85,B 0,C 180,E1 11048.04,E2 11048.04} C_VEL
LIN {X 0,Y 391.839,Z 1061.485,A -85,B 0,C 180,E1 11052.285,E2 11052.285} C_VEL
LIN {X 0,Y 390.326,Z 1078.613,A -85,B 0,C 180,E1 11056.542,E2 11056.542} C_VEL
LIN {X 0,Y 389.777,Z 1089.526,A -85,B 0,C 180,E1 11060.423,E2 11060.423} C_VEL
LIN {X 0,Y 387.217,Z 1093.053,A -85,B 0,C 180,E1 11062.251,E2 11062.251} C_VEL
LIN {X 0,Y 381.968,Z 1096.446,A -85,B 0,C 180,E1 11065.07,E2 11065.07} C_VEL
LIN {X 0,Y 381.893,Z 1096.803,A -85,B 0,C 180,E1 11065.397,E2 11065.397} C_VEL
LIN {X 0,Y 381.989,Z 1099.223,A -85,B 0,C 180,E1 11070.001,E2 11070.001} C_VEL
LIN {X 0,Y 381.893,Z 1096.836,A -85,B 0,C 180,E1 11074.549,E2 11074.549} C_VEL
LIN {X 0,Y 381.952,Z 1089.663,A -85,B 0,C 180,E1 11079.124,E2 11079.124} C_VEL
LIN {X 0,Y 382.58,Z 1076.11,A -85,B 0,C 180,E1 11084.12,E2 11084.12} C_VEL
LIN {X 0,Y 384.536,Z 1057.106,A -85,B 0,C 180,E1 11088.772,E2 11088.772} C_VEL
LIN {X 0,Y 387.733,Z 1032.794,A -85,B 0,C 180,E1 11092.986,E2 11092.986} C_VEL
LIN {X 0,Y 391.92,Z 1003.897,A -85,B 0,C 180,E1 11096.532,E2 11096.532} C_VEL
LIN {X 0,Y 396.169,Z 971.949,A -85,B 0,C 180,E1 11099.216,E2 11099.216} C_VEL
LIN {X 0,Y 399.625,Z 938.687,A -85,B 0,C 180,E1 11100.991,E2 11100.991} C_VEL
LIN {X 0,Y 400.67,Z 912.424,A -85,B 0,C 180,E1 11101.855,E2 11101.855} C_VEL
LIN {X 0,Y 388.087,Z 877.157,A -85,B 0,C 180,E1 11103.724,E2 11103.724} C_VEL
LIN {X 0,Y 379.415,Z 857.28,A -85,B 0,C 180,E1 11105.077,E2 11105.077} C_VEL
LIN {X 0,Y 379.194,Z 857.28,A -85,B 0,C 180,E1 11112.75,E2 11112.75} C_VEL
LIN {X 0,Y 379.253,Z 857.28,A -85,B 0,C 180,E1 11120.283,E2 11120.283} C_VEL
LIN {X 0,Y 379.474,Z 857.28,A -85,B 0,C 180,E1 11126.919,E2 11126.919} C_VEL
LIN {X 0,Y 379.656,Z 857.28,A -85,B 0,C 180,E1 11133.96,E2 11133.96} C_VEL
LIN {X 0,Y 379.93,Z 857.28,A -85,B 0,C 180,E1 11141.386,E2 11141.386} C_VEL
LIN {X 0,Y 380.095,Z 857.28,A -85,B 0,C 180,E1 11148.487,E2 11148.487} C_VEL
LIN {X 0,Y 380.563,Z 857.28,A -85,B 0,C 180,E1 11155.409,E2 11155.409} C_VEL
LIN {X 0,Y 380.756,Z 857.28,A -85,B 0,C 180,E1 11162.249,E2 11162.249} C_VEL
LIN {X 0,Y 380.336,Z 857.28,A -85,B 0,C 180,E1 11169.129,E2 11169.129} C_VEL
LIN {X 0,Y 380.047,Z 857.28,A -85,B 0,C 180,E1 11176.155,E2 11176.155} C_VEL
LIN {X 0,Y 379.706,Z 857.28,A -85,B 0,C 180,E1 11183.489,E2 11183.489} C_VEL
LIN {X 0,Y 379.41,Z 857.28,A -85,B 0,C 180,E1 11191.201,E2 11191.201} C_VEL
LIN {X 0,Y 379.241,Z 857.28,A -85,B 0,C 180,E1 11197.014,E2 11197.014} C_VEL
LIN {X 0,Y 379.199,Z 857.28,A -85,B 0,C 180,E1 11204.051,E2 11204.051} C_VEL
LIN {X 0,Y 379.42,Z 857.28,A -85,B 0,C 180,E1 11206.304,E2 11206.304} C_VEL
LIN {X 0,Y 390.385,Z 886.919,A -85,B 0,C 180,E1 11209.065,E2 11209.065} C_VEL
LIN {X 0,Y 395.567,Z 910.319,A -85,B 0,C 180,E1 11211.647,E2 11211.647} C_VEL
LIN {X 0,Y 392.16,Z 933.853,A -85,B 0,C 180,E1 11214.388,E2 11214.388} C_VEL
LIN {X 0,Y 388.689,Z 954.156,A -85,B 0,C 180,E1 11217.884,E2 11217.884} C_VEL
LIN {X 0,Y 385.853,Z 969.513,A -85,B 0,C 180,E1 11221.908,E2 11221.908} C_VEL
LIN {X 0,Y 384.107,Z 978.675,A -85,B 0,C 180,E1 11225.775,E2 11225.775} C_VEL
LIN {X 0,Y 383.172,Z 983.075,A -85,B 0,C 180,E1 11229.167,E2 11229.167} C_VEL
LIN {X 0,Y 382.7,Z 984.07,A -85,B 0,C 180,E1 11233.921,E2 11233.921} C_VEL
LIN {X 0,Y 383.353,Z 979.215,A -85,B 0,C 180,E1 11238.61,E2 11238.61} C_VEL
LIN {X 0,Y 384.586,Z 969.97,A -85,B 0,C 180,E1 11242.648,E2 11242.648} C_VEL
LIN {X 0,Y 386.617,Z 955.389,A -85,B 0,C 180,E1 11246.568,E2 11246.568} C_VEL
LIN {X 0,Y 389.179,Z 936.312,A -85,B 0,C 180,E1 11249.999,E2 11249.999} C_VEL
LIN {X 0,Y 392.091,Z 912.557,A -85,B 0,C 180,E1 11252.904,E2 11252.904} C_VEL
LIN {X 0,Y 391.868,Z 901.443,A -85,B 0,C 180,E1 11254.015,E2 11254.015} C_VEL
LIN {X 0,Y 385.93,Z 875.306,A -85,B 0,C 180,E1 11256.335,E2 11256.335} C_VEL
LIN {X 0,Y 380.446,Z 857.28,A -85,B 0,C 180,E1 11257.618,E2 11257.618} C_VEL
LIN {X 0,Y 380.168,Z 857.28,A -85,B 0,C 180,E1 11263.824,E2 11263.824} C_VEL
LIN {X 0,Y 379.781,Z 857.28,A -85,B 0,C 180,E1 11271.026,E2 11271.026} C_VEL
LIN {X 0,Y 379.449,Z 857.28,A -85,B 0,C 180,E1 11278.723,E2 11278.723} C_VEL
LIN {X 0,Y 379.35,Z 857.28,A -85,B 0,C 180,E1 11283.97,E2 11283.97} C_VEL
LIN {X 0,Y 379.193,Z 857.28,A -85,B 0,C 180,E1 11290.729,E2 11290.729} C_VEL
LIN {X 0,Y 379.51,Z 857.564,A -85,B 0,C 180,E1 11295.367,E2 11295.367} C_VEL
LIN {X 0,Y 386.744,Z 885.664,A -85,B 0,C 180,E1 11297.02,E2 11297.02} C_VEL
LIN {X 0,Y 389.652,Z 905.237,A -85,B 0,C 180,E1 11298.623,E2 11298.623} C_VEL
LIN {X 0,Y 387.649,Z 930.359,A -85,B 0,C 180,E1 11301.222,E2 11301.222} C_VEL
LIN {X 0,Y 385.707,Z 951.231,A -85,B 0,C 180,E1 11304.447,E2 11304.447} C_VEL
LIN {X 0,Y 384.227,Z 968.151,A -85,B 0,C 180,E1 11308.404,E2 11308.404} C_VEL
LIN {X 0,Y 383.241,Z 978.826,A -85,B 0,C 180,E1 11312.507,E2 11312.507} C_VEL
LIN {X 0,Y 382.768,Z 984.054,A -85,B 0,C 180,E1 11316.741,E2 11316.741} C_VEL
LIN {X 0,Y 382.865,Z 984.632,A -85,B 0,C 180,E1 11319.191,E2 11319.191} C_VEL
LIN {X 0,Y 383.471,Z 982.1,A -85,B 0,C 180,E1 11322.813,E2 11322.813} C_VEL
LIN {X 0,Y 384.703,Z 974.13,A -85,B 0,C 180,E1 11326.956,E2 11326.956} C_VEL
LIN {X 0,Y 386.52,Z 960.928,A -85,B 0,C 180,E1 11330.772,E2 11330.772} C_VEL
LIN {X 0,Y 388.715,Z 942.695,A -85,B 0,C 180,E1 11334.187,E2 11334.187} C_VEL
LIN {X 0,Y 390.95,Z 920.396,A -85,B 0,C 180,E1 11336.977,E2 11336.977} C_VEL
LIN {X 0,Y 391.862,Z 899.11,A -85,B 0,C 180,E1 11338.829,E2 11338.829} C_VEL
LIN {X 0,Y 385.695,Z 872.068,A -85,B 0,C 180,E1 11340.837,E2 11340.837} C_VEL
LIN {X 0,Y 380.76,Z 857.28,A -85,B 0,C 180,E1 11341.737,E2 11341.737} C_VEL
LIN {X 0,Y 380.351,Z 857.28,A -85,B 0,C 180,E1 11349.188,E2 11349.188} C_VEL
LIN {X 0,Y 380.034,Z 857.28,A -85,B 0,C 180,E1 11356.217,E2 11356.217} C_VEL
LIN {X 0,Y 379.735,Z 857.28,A -85,B 0,C 180,E1 11363.519,E2 11363.519} C_VEL
LIN {X 0,Y 379.449,Z 857.28,A -85,B 0,C 180,E1 11371.266,E2 11371.266} C_VEL
LIN {X 0,Y 379.278,Z 857.28,A -85,B 0,C 180,E1 11377.024,E2 11377.024} C_VEL
LIN {X 0,Y 379.23,Z 857.28,A -85,B 0,C 180,E1 11384.058,E2 11384.058} C_VEL
LIN {X 0,Y 379.266,Z 857.28,A -85,B 0,C 180,E1 11390.303,E2 11390.303} C_VEL
LIN {X 0,Y 379.557,Z 857.28,A -85,B 0,C 180,E1 11396.001,E2 11396.001} C_VEL
LIN {X 0,Y 399.811,Z 913.735,A -85,B 0,C 180,E1 11398.595,E2 11398.595} C_VEL
LIN {X 0,Y 397.641,Z 949.417,A -85,B 0,C 180,E1 11399.823,E2 11399.823} C_VEL
LIN {X 0,Y 394.252,Z 981.411,A -85,B 0,C 180,E1 11401.756,E2 11401.756} C_VEL
LIN {X 0,Y 390.315,Z 1012.217,A -85,B 0,C 180,E1 11404.589,E2 11404.589} C_VEL
LIN {X 0,Y 386.668,Z 1039.325,A -85,B 0,C 180,E1 11408.162,E2 11408.162} C_VEL
LIN {X 0,Y 383.819,Z 1062.651,A -85,B 0,C 180,E1 11412.496,E2 11412.496} C_VEL
LIN {X 0,Y 382.379,Z 1079.12,A -85,B 0,C 180,E1 11416.84,E2 11416.84} C_VEL
LIN {X 0,Y 381.895,Z 1091.619,A -85,B 0,C 180,E1 11421.846,E2 11421.846} C_VEL
LIN {X 0,Y 381.893,Z 1096.803,A -85,B 0,C 180,E1 11425.397,E2 11425.397} C_VEL
LIN {X 0,Y 379.514,Z 1098.142,A -85,B 0,C 180,E1 11427.32,E2 11427.32} C_VEL
LIN {X 0,Y 374.096,Z 1097.882,A -85,B 0,C 180,E1 11430.577,E2 11430.577} C_VEL
LIN {X 0,Y 374.068,Z 1094.333,A -85,B 0,C 180,E1 11435.809,E2 11435.809} C_VEL
LIN {X 0,Y 374.124,Z 1085.933,A -85,B 0,C 180,E1 11440.494,E2 11440.494} C_VEL
LIN {X 0,Y 375.113,Z 1071.148,A -85,B 0,C 180,E1 11445.51,E2 11445.51} C_VEL
LIN {X 0,Y 377.406,Z 1051.036,A -85,B 0,C 180,E1 11450.161,E2 11450.161} C_VEL
LIN {X 0,Y 381.136,Z 1025.947,A -85,B 0,C 180,E1 11454.285,E2 11454.285} C_VEL
LIN {X 0,Y 385.5,Z 997.005,A -85,B 0,C 180,E1 11457.643,E2 11457.643} C_VEL
LIN {X 0,Y 389.878,Z 965.09,A -85,B 0,C 180,E1 11460.161,E2 11460.161} C_VEL
LIN {X 0,Y 393.258,Z 932.399,A -85,B 0,C 180,E1 11461.787,E2 11461.787} C_VEL
LIN {X 0,Y 393.569,Z 913.323,A -85,B 0,C 180,E1 11462.437,E2 11462.437} C_VEL
LIN {X 0,Y 380.983,Z 878.392,A -85,B 0,C 180,E1 11464.386,E2 11464.386} C_VEL
LIN {X 0,Y 371.447,Z 857.28,A -85,B 0,C 180,E1 11465.988,E2 11465.988} C_VEL
LIN {X 0,Y 371.294,Z 857.28,A -85,B 0,C 180,E1 11472.759,E2 11472.759} C_VEL
LIN {X 0,Y 371.36,Z 857.28,A -85,B 0,C 180,E1 11479.264,E2 11479.264} C_VEL
LIN {X 0,Y 371.393,Z 857.28,A -85,B 0,C 180,E1 11485.179,E2 11485.179} C_VEL
LIN {X 0,Y 371.565,Z 857.28,A -85,B 0,C 180,E1 11490.706,E2 11490.706} C_VEL
LIN {X 0,Y 371.764,Z 857.28,A -85,B 0,C 180,E1 11495.945,E2 11495.945} C_VEL
LIN {X 0,Y 372.048,Z 857.28,A -85,B 0,C 180,E1 11503.425,E2 11503.425} C_VEL
LIN {X 0,Y 372.366,Z 857.28,A -85,B 0,C 180,E1 11510.613,E2 11510.613} C_VEL
LIN {X 0,Y 372.901,Z 857.28,A -85,B 0,C 180,E1 11517.644,E2 11517.644} C_VEL
LIN {X 0,Y 372.733,Z 857.28,A -85,B 0,C 180,E1 11524.628,E2 11524.628} C_VEL
LIN {X 0,Y 372.296,Z 857.28,A -85,B 0,C 180,E1 11531.697,E2 11531.697} C_VEL
LIN {X 0,Y 371.982,Z 857.28,A -85,B 0,C 180,E1 11538.963,E2 11538.963} C_VEL
LIN {X 0,Y 371.676,Z 857.28,A -85,B 0,C 180,E1 11546.576,E2 11546.576} C_VEL
LIN {X 0,Y 371.499,Z 857.28,A -85,B 0,C 180,E1 11551.943,E2 11551.943} C_VEL
LIN {X 0,Y 371.255,Z 857.28,A -85,B 0,C 180,E1 11559.205,E2 11559.205} C_VEL
LIN {X 0,Y 371.379,Z 857.329,A -85,B 0,C 180,E1 11565.441,E2 11565.441} C_VEL
LIN {X 0,Y 382.421,Z 885.922,A -85,B 0,C 180,E1 11568.205,E2 11568.205} C_VEL
LIN {X 0,Y 388.316,Z 910.076,A -85,B 0,C 180,E1 11570.951,E2 11570.951} C_VEL
LIN {X 0,Y 385.088,Z 934.559,A -85,B 0,C 180,E1 11573.859,E2 11573.859} C_VEL
LIN {X 0,Y 381.506,Z 954.267,A -85,B 0,C 180,E1 11577.265,E2 11577.265} C_VEL
LIN {X 0,Y 378.431,Z 969.836,A -85,B 0,C 180,E1 11581.306,E2 11581.306} C_VEL
LIN {X 0,Y 376.502,Z 979.48,A -85,B 0,C 180,E1 11585.346,E2 11585.346} C_VEL
LIN {X 0,Y 375.497,Z 983.975,A -85,B 0,C 180,E1 11588.721,E2 11588.721} C_VEL
LIN {X 0,Y 374.876,Z 985.37,A -85,B 0,C 180,E1 11593.576,E2 11593.576} C_VEL
LIN {X 0,Y 375.5,Z 980.903,A -85,B 0,C 180,E1 11598.368,E2 11598.368} C_VEL
LIN {X 0,Y 376.741,Z 972.041,A -85,B 0,C 180,E1 11602.494,E2 11602.494} C_VEL
LIN {X 0,Y 378.835,Z 957.587,A -85,B 0,C 180,E1 11606.584,E2 11606.584} C_VEL
LIN {X 0,Y 381.663,Z 937.674,A -85,B 0,C 180,E1 11610.283,E2 11610.283} C_VEL
LIN {X 0,Y 384.678,Z 914.084,A -85,B 0,C 180,E1 11613.243,E2 11613.243} C_VEL
LIN {X 0,Y 384.447,Z 903.116,A -85,B 0,C 180,E1 11614.375,E2 11614.375} C_VEL
LIN {X 0,Y 378.619,Z 877.078,A -85,B 0,C 180,E1 11616.765,E2 11616.765} C_VEL
LIN {X 0,Y 372.515,Z 857.28,A -85,B 0,C 180,E1 11618.251,E2 11618.251} C_VEL
LIN {X 0,Y 372.246,Z 857.28,A -85,B 0,C 180,E1 11624.125,E2 11624.125} C_VEL
LIN {X 0,Y 371.809,Z 857.28,A -85,B 0,C 180,E1 11631.499,E2 11631.499} C_VEL
LIN {X 0,Y 371.597,Z 857.28,A -85,B 0,C 180,E1 11636.627,E2 11636.627} C_VEL
LIN {X 0,Y 371.437,Z 857.28,A -85,B 0,C 180,E1 11641.999,E2 11641.999} C_VEL
LIN {X 0,Y 371.248,Z 857.28,A -85,B 0,C 180,E1 11649.283,E2 11649.283} C_VEL
LIN {X 0,Y 371.587,Z 857.623,A -85,B 0,C 180,E1 11654.936,E2 11654.936} C_VEL
LIN {X 0,Y 378.991,Z 886.057,A -85,B 0,C 180,E1 11656.627,E2 11656.627} C_VEL
LIN {X 0,Y 382.109,Z 906.258,A -85,B 0,C 180,E1 11658.308,E2 11658.308} C_VEL
LIN {X 0,Y 379.975,Z 932.294,A -85,B 0,C 180,E1 11661.068,E2 11661.068} C_VEL
LIN {X 0,Y 377.918,Z 953.372,A -85,B 0,C 180,E1 11664.446,E2 11664.446} C_VEL
LIN {X 0,Y 376.515,Z 968.523,A -85,B 0,C 180,E1 11668.051,E2 11668.051} C_VEL
LIN {X 0,Y 375.516,Z 978.91,A -85,B 0,C 180,E1 11671.896,E2 11671.896} C_VEL
LIN {X 0,Y 374.983,Z 984.93,A -85,B 0,C 180,E1 11676.229,E2 11676.229} C_VEL
LIN {X 0,Y 375.036,Z 985.869,A -85,B 0,C 180,E1 11678.736,E2 11678.736} C_VEL
LIN {X 0,Y 375.635,Z 983.932,A -85,B 0,C 180,E1 11682.471,E2 11682.471} C_VEL
LIN {X 0,Y 376.84,Z 976.654,A -85,B 0,C 180,E1 11686.679,E2 11686.679} C_VEL
LIN {X 0,Y 378.878,Z 963.288,A -85,B 0,C 180,E1 11690.836,E2 11690.836} C_VEL
LIN {X 0,Y 381.209,Z 944.93,A -85,B 0,C 180,E1 11694.411,E2 11694.411} C_VEL
LIN {X 0,Y 383.648,Z 922.254,A -85,B 0,C 180,E1 11697.344,E2 11697.344} C_VEL
LIN {X 0,Y 384.553,Z 900.168,A -85,B 0,C 180,E1 11699.324,E2 11699.324} C_VEL
LIN {X 0,Y 378.407,Z 873.186,A -85,B 0,C 180,E1 11701.385,E2 11701.385} C_VEL
LIN {X 0,Y 372.826,Z 857.28,A -85,B 0,C 180,E1 11702.502,E2 11702.502} C_VEL
LIN {X 0,Y 372.413,Z 857.28,A -85,B 0,C 180,E1 11709.385,E2 11709.385} C_VEL
LIN {X 0,Y 372.12,Z 857.28,A -85,B 0,C 180,E1 11716.572,E2 11716.572} C_VEL
LIN {X 0,Y 371.756,Z 857.28,A -85,B 0,C 180,E1 11724.056,E2 11724.056} C_VEL
LIN {X 0,Y 371.525,Z 857.28,A -85,B 0,C 180,E1 11732.011,E2 11732.011} C_VEL
LIN {X 0,Y 371.3,Z 857.28,A -85,B 0,C 180,E1 11739.216,E2 11739.216} C_VEL
LIN {X 0,Y 371.34,Z 857.28,A -85,B 0,C 180,E1 11746.121,E2 11746.121} C_VEL
LIN {X 0,Y 371.32,Z 857.28,A -85,B 0,C 180,E1 11752.293,E2 11752.293} C_VEL
LIN {X 0,Y 371.586,Z 857.28,A -85,B 0,C 180,E1 11755.385,E2 11755.385} C_VEL
LIN {X 0,Y 392.362,Z 914.196,A -85,B 0,C 180,E1 11758.112,E2 11758.112} C_VEL
LIN {X 0,Y 390.451,Z 948.221,A -85,B 0,C 180,E1 11759.33,E2 11759.33} C_VEL
LIN {X 0,Y 386.818,Z 981.1,A -85,B 0,C 180,E1 11761.349,E2 11761.349} C_VEL
LIN {X 0,Y 382.797,Z 1011.581,A -85,B 0,C 180,E1 11764.21,E2 11764.21} C_VEL
LIN {X 0,Y 379.124,Z 1037.647,A -85,B 0,C 180,E1 11767.705,E2 11767.705} C_VEL
LIN {X 0,Y 376.106,Z 1061.184,A -85,B 0,C 180,E1 11772.125,E2 11772.125} C_VEL
LIN {X 0,Y 374.587,Z 1077.775,A -85,B 0,C 180,E1 11776.562,E2 11776.562} C_VEL
LIN {X 0,Y 374.043,Z 1090.009,A -85,B 0,C 180,E1 11781.475,E2 11781.475} C_VEL
LIN {X 0,Y 374.073,Z 1095.677,A -85,B 0,C 180,E1 11785.391,E2 11785.391} C_VEL
LIN {X 0,Y 374.188,Z 1098.045,A -85,B 0,C 180,E1 11790.001,E2 11790.001} C_VEL
LIN {X 0,Y 374.096,Z 1097.882,A -85,B 0,C 180,E1 11790.577,E2 11790.577} C_VEL
LIN {X 0,Y 372.749,Z 1097.416,A -85,B 0,C 180,E1 11791.895,E2 11791.895} C_VEL
LIN {X 0,Y 366.295,Z 1093.695,A -85,B 0,C 180,E1 11795.475,E2 11795.475} C_VEL
LIN {X 0,Y 366.216,Z 1093.298,A -85,B 0,C 180,E1 11795.815,E2 11795.815} C_VEL
LIN {X 0,Y 366.272,Z 1084.774,A -85,B 0,C 180,E1 11800.721,E2 11800.721} C_VEL
LIN {X 0,Y 367.369,Z 1069.985,A -85,B 0,C 180,E1 11805.846,E2 11805.846} C_VEL
LIN {X 0,Y 369.781,Z 1049.934,A -85,B 0,C 180,E1 11810.587,E2 11810.587} C_VEL
LIN {X 0,Y 373.627,Z 1025.401,A -85,B 0,C 180,E1 11814.716,E2 11814.716} C_VEL
LIN {X 0,Y 378.302,Z 996.304,A -85,B 0,C 180,E1 11818.169,E2 11818.169} C_VEL
LIN {X 0,Y 382.976,Z 963.999,A -85,B 0,C 180,E1 11820.763,E2 11820.763} C_VEL
LIN {X 0,Y 386.49,Z 931.367,A -85,B 0,C 180,E1 11822.402,E2 11822.402} C_VEL
LIN {X 0,Y 386.784,Z 915.456,A -85,B 0,C 180,E1 11822.968,E2 11822.968} C_VEL
LIN {X 0,Y 374.884,Z 882.073,A -85,B 0,C 180,E1 11824.919,E2 11824.919} C_VEL
LIN {X 0,Y 363.463,Z 857.28,A -85,B 0,C 180,E1 11826.865,E2 11826.865} C_VEL
LIN {X 0,Y 363.361,Z 857.28,A -85,B 0,C 180,E1 11831.814,E2 11831.814} C_VEL
LIN {X 0,Y 363.406,Z 857.28,A -85,B 0,C 180,E1 11838.587,E2 11838.587} C_VEL
LIN {X 0,Y 363.425,Z 857.28,A -85,B 0,C 180,E1 11844.3,E2 11844.3} C_VEL
LIN {X 0,Y 363.659,Z 857.28,A -85,B 0,C 180,E1 11850.967,E2 11850.967} C_VEL
LIN {X 0,Y 363.892,Z 857.28,A -85,B 0,C 180,E1 11857.986,E2 11857.986} C_VEL
LIN {X 0,Y 364.118,Z 857.28,A -85,B 0,C 180,E1 11865.527,E2 11865.527} C_VEL
LIN {X 0,Y 364.693,Z 857.28,A -85,B 0,C 180,E1 11872.818,E2 11872.818} C_VEL
LIN {X 0,Y 365.058,Z 857.28,A -85,B 0,C 180,E1 11879.97,E2 11879.97} C_VEL
LIN {X 0,Y 364.66,Z 857.28,A -85,B 0,C 180,E1 11887.122,E2 11887.122} C_VEL
LIN {X 0,Y 364.263,Z 857.28,A -85,B 0,C 180,E1 11894.404,E2 11894.404} C_VEL
LIN {X 0,Y 363.9,Z 857.28,A -85,B 0,C 180,E1 11901.948,E2 11901.948} C_VEL
LIN {X 0,Y 363.6,Z 857.28,A -85,B 0,C 180,E1 11909.93,E2 11909.93} C_VEL
LIN {X 0,Y 363.375,Z 857.28,A -85,B 0,C 180,E1 11917.656,E2 11917.656} C_VEL
LIN {X 0,Y 363.425,Z 857.28,A -85,B 0,C 180,E1 11924.481,E2 11924.481} C_VEL
LIN {X 0,Y 375.221,Z 887.2,A -85,B 0,C 180,E1 11927.541,E2 11927.541} C_VEL
LIN {X 0,Y 381.257,Z 911.94,A -85,B 0,C 180,E1 11930.466,E2 11930.466} C_VEL
LIN {X 0,Y 377.801,Z 936.704,A -85,B 0,C 180,E1 11933.51,E2 11933.51} C_VEL
LIN {X 0,Y 373.864,Z 957.072,A -85,B 0,C 180,E1 11937.202,E2 11937.202} C_VEL
LIN {X 0,Y 370.789,Z 971.598,A -85,B 0,C 180,E1 11941.168,E2 11941.168} C_VEL
LIN {X 0,Y 368.584,Z 981.748,A -85,B 0,C 180,E1 11945.745,E2 11945.745} C_VEL
LIN {X 0,Y 367.279,Z 986.488,A -85,B 0,C 180,E1 11950.743,E2 11950.743} C_VEL
LIN {X 0,Y 367.212,Z 985.298,A -85,B 0,C 180,E1 11955.676,E2 11955.676} C_VEL
LIN {X 0,Y 368.296,Z 978.28,A -85,B 0,C 180,E1 11960.534,E2 11960.534} C_VEL
LIN {X 0,Y 370.026,Z 965.835,A -85,B 0,C 180,E1 11965.011,E2 11965.011} C_VEL
LIN {X 0,Y 372.736,Z 947.627,A -85,B 0,C 180,E1 11969.126,E2 11969.126} C_VEL
LIN {X 0,Y 376,Z 925.55,A -85,B 0,C 180,E1 11972.451,E2 11972.451} C_VEL
LIN {X 0,Y 377.511,Z 907.351,A -85,B 0,C 180,E1 11974.456,E2 11974.456} C_VEL
LIN {X 0,Y 371.96,Z 881.139,A -85,B 0,C 180,E1 11977.013,E2 11977.013} C_VEL
LIN {X 0,Y 364.611,Z 857.28,A -85,B 0,C 180,E1 11978.885,E2 11978.885} C_VEL
LIN {X 0,Y 364.291,Z 857.28,A -85,B 0,C 180,E1 11984.44,E2 11984.44} C_VEL
LIN {X 0,Y 363.829,Z 857.28,A -85,B 0,C 180,E1 11991.995,E2 11991.995} C_VEL
LIN {X 0,Y 363.531,Z 857.28,A -85,B 0,C 180,E1 11999.985,E2 11999.985} C_VEL
LIN {X 0,Y 363.363,Z 857.28,A -85,B 0,C 180,E1 12007.737,E2 12007.737} C_VEL
LIN {X 0,Y 363.628,Z 857.677,A -85,B 0,C 180,E1 12014.485,E2 12014.485} C_VEL
LIN {X 0,Y 371.372,Z 887.141,A -85,B 0,C 180,E1 12016.273,E2 12016.273} C_VEL
LIN {X 0,Y 374.494,Z 908.022,A -85,B 0,C 180,E1 12018.055,E2 12018.055} C_VEL
LIN {X 0,Y 372.307,Z 933.649,A -85,B 0,C 180,E1 12020.842,E2 12020.842} C_VEL
LIN {X 0,Y 370.132,Z 955.258,A -85,B 0,C 180,E1 12024.4,E2 12024.4} C_VEL
LIN {X 0,Y 368.638,Z 970.952,A -85,B 0,C 180,E1 12028.309,E2 12028.309} C_VEL
LIN {X 0,Y 367.642,Z 981.342,A -85,B 0,C 180,E1 12032.503,E2 12032.503} C_VEL
LIN {X 0,Y 367.208,Z 985.653,A -85,B 0,C 180,E1 12035.694,E2 12035.694} C_VEL
LIN {X 0,Y 367.195,Z 987.069,A -85,B 0,C 180,E1 12038.259,E2 12038.259} C_VEL
LIN {X 0,Y 367.596,Z 986.318,A -85,B 0,C 180,E1 12041.32,E2 12041.32} C_VEL
LIN {X 0,Y 368.758,Z 980.449,A -85,B 0,C 180,E1 12045.776,E2 12045.776} C_VEL
LIN {X 0,Y 370.552,Z 969.506,A -85,B 0,C 180,E1 12049.838,E2 12049.838} C_VEL
LIN {X 0,Y 372.988,Z 952.81,A -85,B 0,C 180,E1 12053.674,E2 12053.674} C_VEL
LIN {X 0,Y 375.614,Z 931.68,A -85,B 0,C 180,E1 12056.854,E2 12056.854} C_VEL
LIN {X 0,Y 377.915,Z 907.047,A -85,B 0,C 180,E1 12059.312,E2 12059.312} C_VEL
LIN {X 0,Y 372.997,Z 880.624,A -85,B 0,C 180,E1 12061.511,E2 12061.511} C_VEL
LIN {X 0,Y 364.875,Z 857.28,A -85,B 0,C 180,E1 12063.151,E2 12063.151} C_VEL
LIN {X 0,Y 364.473,Z 857.28,A -85,B 0,C 180,E1 12069.592,E2 12069.592} C_VEL
LIN {X 0,Y 364.158,Z 857.28,A -85,B 0,C 180,E1 12077.007,E2 12077.007} C_VEL
LIN {X 0,Y 363.8,Z 857.28,A -85,B 0,C 180,E1 12084.616,E2 12084.616} C_VEL
LIN {X 0,Y 363.645,Z 857.28,A -85,B 0,C 180,E1 12089.997,E2 12089.997} C_VEL
LIN {X 0,Y 363.401,Z 857.28,A -85,B 0,C 180,E1 12097.664,E2 12097.664} C_VEL
LIN {X 0,Y 363.377,Z 857.28,A -85,B 0,C 180,E1 12105.118,E2 12105.118} C_VEL
LIN {X 0,Y 363.441,Z 857.28,A -85,B 0,C 180,E1 12112.347,E2 12112.347} C_VEL
LIN {X 0,Y 363.669,Z 857.28,A -85,B 0,C 180,E1 12114.762,E2 12114.762} C_VEL
LIN {X 0,Y 385.267,Z 916.232,A -85,B 0,C 180,E1 12117.682,E2 12117.682} C_VEL
LIN {X 0,Y 382.999,Z 950.207,A -85,B 0,C 180,E1 12118.974,E2 12118.974} C_VEL
LIN {X 0,Y 379.219,Z 982.22,A -85,B 0,C 180,E1 12121.047,E2 12121.047} C_VEL
LIN {X 0,Y 375.095,Z 1012.126,A -85,B 0,C 180,E1 12123.963,E2 12123.963} C_VEL
LIN {X 0,Y 371.042,Z 1039.651,A -85,B 0,C 180,E1 12127.825,E2 12127.825} C_VEL
LIN {X 0,Y 368.088,Z 1062.25,A -85,B 0,C 180,E1 12132.341,E2 12132.341} C_VEL
LIN {X 0,Y 366.618,Z 1078.392,A -85,B 0,C 180,E1 12136.925,E2 12136.925} C_VEL
LIN {X 0,Y 366.218,Z 1090.472,A -85,B 0,C 180,E1 12142.279,E2 12142.279} C_VEL
LIN {X 0,Y 366.251,Z 1094.434,A -85,B 0,C 180,E1 12145.258,E2 12145.258} C_VEL
LIN {X 0,Y 366.373,Z 1096.863,A -85,B 0,C 180,E1 12150.001,E2 12150.001} C_VEL
LIN {X 0,Y 366.249,Z 1094.511,A -85,B 0,C 180,E1 12154.743,E2 12154.743} C_VEL
LIN {X 0,Y 366.216,Z 1093.298,A -85,B 0,C 180,E1 12155.815,E2 12155.815} C_VEL
LIN {X 0,Y 363.737,Z 1090.375,A -85,B 0,C 180,E1 12157.786,E2 12157.786} C_VEL
LIN {X 0,Y 358.498,Z 1084.265,A -85,B 0,C 180,E1 12160.684,E2 12160.684} C_VEL
LIN {X 0,Y 358.424,Z 1083.487,A -85,B 0,C 180,E1 12161.015,E2 12161.015} C_VEL
LIN {X 0,Y 359.758,Z 1067.809,A -85,B 0,C 180,E1 12166.505,E2 12166.505} C_VEL
LIN {X 0,Y 362.581,Z 1046.829,A -85,B 0,C 180,E1 12171.432,E2 12171.432} C_VEL
LIN {X 0,Y 366.82,Z 1021.162,A -85,B 0,C 180,E1 12175.684,E2 12175.684} C_VEL
LIN {X 0,Y 371.789,Z 991.736,A -85,B 0,C 180,E1 12179.101,E2 12179.101} C_VEL
LIN {X 0,Y 376.618,Z 958.65,A -85,B 0,C 180,E1 12181.67,E2 12181.67} C_VEL
LIN {X 0,Y 380.137,Z 925.359,A -85,B 0,C 180,E1 12183.22,E2 12183.22} C_VEL
LIN {X 0,Y 379.626,Z 915.774,A -85,B 0,C 180,E1 12183.622,E2 12183.622} C_VEL
LIN {X 0,Y 367.902,Z 883.552,A -85,B 0,C 180,E1 12185.632,E2 12185.632} C_VEL
LIN {X 0,Y 355.501,Z 857.28,A -85,B 0,C 180,E1 12187.773,E2 12187.773} C_VEL
LIN {X 0,Y 355.33,Z 857.28,A -85,B 0,C 180,E1 12193.564,E2 12193.564} C_VEL
LIN {X 0,Y 355.421,Z 857.28,A -85,B 0,C 180,E1 12200.263,E2 12200.263} C_VEL
LIN {X 0,Y 355.546,Z 857.28,A -85,B 0,C 180,E1 12206.365,E2 12206.365} C_VEL
LIN {X 0,Y 355.763,Z 857.28,A -85,B 0,C 180,E1 12213.348,E2 12213.348} C_VEL
LIN {X 0,Y 356.065,Z 857.28,A -85,B 0,C 180,E1 12220.088,E2 12220.088} C_VEL
LIN {X 0,Y 356.321,Z 857.28,A -85,B 0,C 180,E1 12227.777,E2 12227.777} C_VEL
LIN {X 0,Y 356.851,Z 857.28,A -85,B 0,C 180,E1 12235.103,E2 12235.103} C_VEL
LIN {X 0,Y 357.168,Z 857.28,A -85,B 0,C 180,E1 12239.969,E2 12239.969} C_VEL
LIN {X 0,Y 356.724,Z 857.28,A -85,B 0,C 180,E1 12247.281,E2 12247.281} C_VEL
LIN {X 0,Y 356.311,Z 857.28,A -85,B 0,C 180,E1 12254.732,E2 12254.732} C_VEL
LIN {X 0,Y 355.952,Z 857.28,A -85,B 0,C 180,E1 12262.465,E2 12262.465} C_VEL
LIN {X 0,Y 355.734,Z 857.28,A -85,B 0,C 180,E1 12267.868,E2 12267.868} C_VEL
LIN {X 0,Y 355.548,Z 857.28,A -85,B 0,C 180,E1 12273.56,E2 12273.56} C_VEL
LIN {X 0,Y 355.343,Z 857.28,A -85,B 0,C 180,E1 12279.917,E2 12279.917} C_VEL
LIN {X 0,Y 355.451,Z 857.28,A -85,B 0,C 180,E1 12283.522,E2 12283.522} C_VEL
LIN {X 0,Y 366.982,Z 885.461,A -85,B 0,C 180,E1 12286.498,E2 12286.498} C_VEL
LIN {X 0,Y 373.563,Z 910.15,A -85,B 0,C 180,E1 12289.478,E2 12289.478} C_VEL
LIN {X 0,Y 373.812,Z 920.455,A -85,B 0,C 180,E1 12290.734,E2 12290.734} C_VEL
LIN {X 0,Y 369.556,Z 944.057,A -85,B 0,C 180,E1 12293.996,E2 12293.996} C_VEL
LIN {X 0,Y 365.479,Z 963.081,A -85,B 0,C 180,E1 12297.943,E2 12297.943} C_VEL
LIN {X 0,Y 362.676,Z 975.455,A -85,B 0,C 180,E1 12301.815,E2 12301.815} C_VEL
LIN {X 0,Y 360.58,Z 984.276,A -85,B 0,C 180,E1 12306.433,E2 12306.433} C_VEL
LIN {X 0,Y 359.563,Z 987.567,A -85,B 0,C 180,E1 12310.313,E2 12310.313} C_VEL
LIN {X 0,Y 359.39,Z 986.625,A -85,B 0,C 180,E1 12315.469,E2 12315.469} C_VEL
LIN {X 0,Y 360.4,Z 980.058,A -85,B 0,C 180,E1 12320.325,E2 12320.325} C_VEL
LIN {X 0,Y 362.129,Z 969.028,A -85,B 0,C 180,E1 12324.601,E2 12324.601} C_VEL
LIN {X 0,Y 364.711,Z 951.988,A -85,B 0,C 180,E1 12328.81,E2 12328.81} C_VEL
LIN {X 0,Y 368.047,Z 930.355,A -85,B 0,C 180,E1 12332.357,E2 12332.357} C_VEL
LIN {X 0,Y 370.288,Z 910.202,A -85,B 0,C 180,E1 12334.69,E2 12334.69} C_VEL
LIN {X 0,Y 364.848,Z 883.634,A -85,B 0,C 180,E1 12337.395,E2 12337.395} C_VEL
LIN {X 0,Y 356.67,Z 857.28,A -85,B 0,C 180,E1 12339.469,E2 12339.469} C_VEL
LIN {X 0,Y 356.205,Z 857.28,A -85,B 0,C 180,E1 12347.309,E2 12347.309} C_VEL
LIN {X 0,Y 355.734,Z 857.28,A -85,B 0,C 180,E1 12355.189,E2 12355.189} C_VEL
LIN {X 0,Y 355.484,Z 857.28,A -85,B 0,C 180,E1 12361.688,E2 12361.688} C_VEL
LIN {X 0,Y 355.421,Z 857.28,A -85,B 0,C 180,E1 12366.611,E2 12366.611} C_VEL
LIN {X 0,Y 355.648,Z 857.52,A -85,B 0,C 180,E1 12374.021,E2 12374.021} C_VEL
LIN {X 0,Y 363.247,Z 886.293,A -85,B 0,C 180,E1 12375.758,E2 12375.758} C_VEL
LIN {X 0,Y 366.961,Z 908.876,A -85,B 0,C 180,E1 12377.711,E2 12377.711} C_VEL
LIN {X 0,Y 364.816,Z 933.47,A -85,B 0,C 180,E1 12380.402,E2 12380.402} C_VEL
LIN {X 0,Y 362.655,Z 954.254,A -85,B 0,C 180,E1 12383.769,E2 12383.769} C_VEL
LIN {X 0,Y 361.054,Z 969.945,A -85,B 0,C 180,E1 12387.528,E2 12387.528} C_VEL
LIN {X 0,Y 359.875,Z 981.835,A -85,B 0,C 180,E1 12392.068,E2 12392.068} C_VEL
LIN {X 0,Y 359.443,Z 986.325,A -85,B 0,C 180,E1 12395.133,E2 12395.133} C_VEL
LIN {X 0,Y 359.365,Z 988.185,A -85,B 0,C 180,E1 12397.955,E2 12397.955} C_VEL
LIN {X 0,Y 359.612,Z 988.131,A -85,B 0,C 180,E1 12400.358,E2 12400.358} C_VEL
LIN {X 0,Y 360.73,Z 983.744,A -85,B 0,C 180,E1 12404.874,E2 12404.874} C_VEL
LIN {X 0,Y 362.512,Z 973.835,A -85,B 0,C 180,E1 12409.206,E2 12409.206} C_VEL
LIN {X 0,Y 364.965,Z 958.384,A -85,B 0,C 180,E1 12413.228,E2 12413.228} C_VEL
LIN {X 0,Y 367.789,Z 938.06,A -85,B 0,C 180,E1 12416.639,E2 12416.639} C_VEL
LIN {X 0,Y 370.383,Z 914.362,A -85,B 0,C 180,E1 12419.298,E2 12419.298} C_VEL
LIN {X 0,Y 370.103,Z 902.544,A -85,B 0,C 180,E1 12420.371,E2 12420.371} C_VEL
LIN {X 0,Y 364.2,Z 876.652,A -85,B 0,C 180,E1 12422.504,E2 12422.504} C_VEL
LIN {X 0,Y 356.916,Z 857.28,A -85,B 0,C 180,E1 12423.937,E2 12423.937} C_VEL
LIN {X 0,Y 356.535,Z 857.28,A -85,B 0,C 180,E1 12429.807,E2 12429.807} C_VEL
LIN {X 0,Y 356.231,Z 857.28,A -85,B 0,C 180,E1 12437.334,E2 12437.334} C_VEL
LIN {X 0,Y 355.804,Z 857.28,A -85,B 0,C 180,E1 12445.207,E2 12445.207} C_VEL
LIN {X 0,Y 355.551,Z 857.28,A -85,B 0,C 180,E1 12451.607,E2 12451.607} C_VEL
LIN {X 0,Y 355.473,Z 857.28,A -85,B 0,C 180,E1 12456.626,E2 12456.626} C_VEL
LIN {X 0,Y 355.35,Z 857.28,A -85,B 0,C 180,E1 12463.587,E2 12463.587} C_VEL
LIN {X 0,Y 355.446,Z 857.28,A -85,B 0,C 180,E1 12470.288,E2 12470.288} C_VEL
LIN {X 0,Y 355.681,Z 857.654,A -85,B 0,C 180,E1 12474.129,E2 12474.129} C_VEL
LIN {X 0,Y 378.107,Z 918.371,A -85,B 0,C 180,E1 12477.252,E2 12477.252} C_VEL
LIN {X 0,Y 375.442,Z 952.586,A -85,B 0,C 180,E1 12478.636,E2 12478.636} C_VEL
LIN {X 0,Y 371.438,Z 984.703,A -85,B 0,C 180,E1 12480.847,E2 12480.847} C_VEL
LIN {X 0,Y 367.056,Z 1015.002,A -85,B 0,C 180,E1 12484.007,E2 12484.007} C_VEL
LIN {X 0,Y 362.992,Z 1041.421,A -85,B 0,C 180,E1 12487.952,E2 12487.952} C_VEL
LIN {X 0,Y 360.098,Z 1063.321,A -85,B 0,C 180,E1 12492.576,E2 12492.576} C_VEL
LIN {X 0,Y 358.641,Z 1078.964,A -85,B 0,C 180,E1 12497.356,E2 12497.356} C_VEL
LIN {X 0,Y 358.394,Z 1090.181,A -85,B 0,C 180,E1 12502.72,E2 12502.72} C_VEL
LIN {X 0,Y 358.398,Z 1095.012,A -85,B 0,C 180,E1 12507.58,E2 12507.58} C_VEL
LIN {X 0,Y 358.558,Z 1095.679,A -85,B 0,C 180,E1 12510.001,E2 12510.001} C_VEL
LIN {X 0,Y 358.417,Z 1093.356,A -85,B 0,C 180,E1 12514.847,E2 12514.847} C_VEL
LIN {X 0,Y 358.392,Z 1084.911,A -85,B 0,C 180,E1 12520.344,E2 12520.344} C_VEL
LIN {X 0,Y 358.424,Z 1083.487,A -85,B 0,C 180,E1 12521.015,E2 12521.015} C_VEL
LIN {X 0,Y 354.812,Z 1076.92,A -85,B 0,C 180,E1 12523.564,E2 12523.564} C_VEL
LIN {X 0,Y 351.639,Z 1069.304,A -85,B 0,C 180,E1 12526.086,E2 12526.086} C_VEL
LIN {X 0,Y 354.219,Z 1050.272,A -85,B 0,C 180,E1 12530.977,E2 12530.977} C_VEL
LIN {X 0,Y 358.366,Z 1026.335,A -85,B 0,C 180,E1 12535.327,E2 12535.327} C_VEL
LIN {X 0,Y 363.534,Z 997.914,A -85,B 0,C 180,E1 12538.981,E2 12538.981} C_VEL
LIN {X 0,Y 368.691,Z 966.32,A -85,B 0,C 180,E1 12541.748,E2 12541.748} C_VEL
LIN {X 0,Y 372.692,Z 934.039,A -85,B 0,C 180,E1 12543.519,E2 12543.519} C_VEL
LIN {X 0,Y 373.143,Z 918.692,A -85,B 0,C 180,E1 12544.15,E2 12544.15} C_VEL
LIN {X 0,Y 362.506,Z 888.514,A -85,B 0,C 180,E1 12546.115,E2 12546.115} C_VEL
LIN {X 0,Y 347.568,Z 857.28,A -85,B 0,C 180,E1 12548.82,E2 12548.82} C_VEL
LIN {X 0,Y 347.368,Z 857.28,A -85,B 0,C 180,E1 12555.761,E2 12555.761} C_VEL
LIN {X 0,Y 347.457,Z 857.28,A -85,B 0,C 180,E1 12562.385,E2 12562.385} C_VEL
LIN {X 0,Y 347.656,Z 857.28,A -85,B 0,C 180,E1 12568.47,E2 12568.47} C_VEL
LIN {X 0,Y 347.88,Z 857.28,A -85,B 0,C 180,E1 12576.064,E2 12576.064} C_VEL
LIN {X 0,Y 348.242,Z 857.28,A -85,B 0,C 180,E1 12583.043,E2 12583.043} C_VEL
LIN {X 0,Y 348.539,Z 857.28,A -85,B 0,C 180,E1 12589.965,E2 12589.965} C_VEL
LIN {X 0,Y 349.181,Z 857.28,A -85,B 0,C 180,E1 12597.484,E2 12597.484} C_VEL
LIN {X 0,Y 349,Z 857.28,A -85,B 0,C 180,E1 12603.773,E2 12603.773} C_VEL
LIN {X 0,Y 348.596,Z 857.28,A -85,B 0,C 180,E1 12609.968,E2 12609.968} C_VEL
LIN {X 0,Y 348.275,Z 857.28,A -85,B 0,C 180,E1 12617.676,E2 12617.676} C_VEL
LIN {X 0,Y 347.861,Z 857.28,A -85,B 0,C 180,E1 12625.754,E2 12625.754} C_VEL
LIN {X 0,Y 347.677,Z 857.28,A -85,B 0,C 180,E1 12631.453,E2 12631.453} C_VEL
LIN {X 0,Y 347.368,Z 857.28,A -85,B 0,C 180,E1 12638.318,E2 12638.318} C_VEL
LIN {X 0,Y 347.469,Z 857.499,A -85,B 0,C 180,E1 12642.473,E2 12642.473} C_VEL
LIN {X 0,Y 359.951,Z 887.126,A -85,B 0,C 180,E1 12645.796,E2 12645.796} C_VEL
LIN {X 0,Y 366.515,Z 912.115,A -85,B 0,C 180,E1 12648.941,E2 12648.941} C_VEL
LIN {X 0,Y 366.923,Z 921.764,A -85,B 0,C 180,E1 12650.177,E2 12650.177} C_VEL
LIN {X 0,Y 362.617,Z 944.459,A -85,B 0,C 180,E1 12653.357,E2 12653.357} C_VEL
LIN {X 0,Y 358.332,Z 963.467,A -85,B 0,C 180,E1 12657.308,E2 12657.308} C_VEL
LIN {X 0,Y 355.061,Z 976.925,A -85,B 0,C 180,E1 12661.591,E2 12661.591} C_VEL
LIN {X 0,Y 352.954,Z 985.116,A -85,B 0,C 180,E1 12665.95,E2 12665.95} C_VEL
LIN {X 0,Y 351.631,Z 989.058,A -85,B 0,C 180,E1 12671.143,E2 12671.143} C_VEL
LIN {X 0,Y 351.695,Z 986.932,A -85,B 0,C 180,E1 12676.471,E2 12676.471} C_VEL
LIN {X 0,Y 353.026,Z 978.833,A -85,B 0,C 180,E1 12681.585,E2 12681.585} C_VEL
LIN {X 0,Y 354.914,Z 966.158,A -85,B 0,C 180,E1 12686.015,E2 12686.015} C_VEL
LIN {X 0,Y 357.891,Z 948.572,A -85,B 0,C 180,E1 12689.999,E2 12689.999} C_VEL
LIN {X 0,Y 361.449,Z 926.019,A -85,B 0,C 180,E1 12693.451,E2 12693.451} C_VEL
LIN {X 0,Y 362.744,Z 911.004,A -85,B 0,C 180,E1 12695.171,E2 12695.171} C_VEL
LIN {X 0,Y 357.609,Z 885.428,A -85,B 0,C 180,E1 12697.852,E2 12697.852} C_VEL
LIN {X 0,Y 348.646,Z 857.28,A -85,B 0,C 180,E1 12700.161,E2 12700.161} C_VEL
LIN {X 0,Y 348.25,Z 857.28,A -85,B 0,C 180,E1 12707.717,E2 12707.717} C_VEL
LIN {X 0,Y 347.777,Z 857.28,A -85,B 0,C 180,E1 12715.807,E2 12715.807} C_VEL
LIN {X 0,Y 347.607,Z 857.28,A -85,B 0,C 180,E1 12721.512,E2 12721.512} C_VEL
LIN {X 0,Y 347.353,Z 857.28,A -85,B 0,C 180,E1 12728.399,E2 12728.399} C_VEL
LIN {X 0,Y 347.667,Z 857.292,A -85,B 0,C 180,E1 12733.535,E2 12733.535} C_VEL
LIN {X 0,Y 355.411,Z 886.325,A -85,B 0,C 180,E1 12735.307,E2 12735.307} C_VEL
LIN {X 0,Y 359.51,Z 908.987,A -85,B 0,C 180,E1 12737.293,E2 12737.293} C_VEL
LIN {X 0,Y 357.201,Z 934.397,A -85,B 0,C 180,E1 12740.102,E2 12740.102} C_VEL
LIN {X 0,Y 354.914,Z 955.767,A -85,B 0,C 180,E1 12743.639,E2 12743.639} C_VEL
LIN {X 0,Y 353.22,Z 972.033,A -85,B 0,C 180,E1 12747.681,E2 12747.681} C_VEL
LIN {X 0,Y 352.11,Z 982.608,A -85,B 0,C 180,E1 12751.82,E2 12751.82} C_VEL
LIN {X 0,Y 351.555,Z 988.275,A -85,B 0,C 180,E1 12755.972,E2 12755.972} C_VEL
LIN {X 0,Y 351.953,Z 989.076,A -85,B 0,C 180,E1 12761.157,E2 12761.157} C_VEL
LIN {X 0,Y 353.271,Z 983.92,A -85,B 0,C 180,E1 12765.772,E2 12765.772} C_VEL
LIN {X 0,Y 355.37,Z 972.998,A -85,B 0,C 180,E1 12770.224,E2 12770.224} C_VEL
LIN {X 0,Y 358.036,Z 957.124,A -85,B 0,C 180,E1 12774.144,E2 12774.144} C_VEL
LIN {X 0,Y 360.948,Z 936.738,A -85,B 0,C 180,E1 12777.477,E2 12777.477} C_VEL
LIN {X 0,Y 363.687,Z 911.68,A -85,B 0,C 180,E1 12780.164,E2 12780.164} C_VEL
LIN {X 0,Y 359.652,Z 886.626,A -85,B 0,C 180,E1 12782.443,E2 12782.443} C_VEL
LIN {X 0,Y 350.239,Z 861.505,A -85,B 0,C 180,E1 12784.459,E2 12784.459} C_VEL
LIN {X 0,Y 349.047,Z 857.28,A -85,B 0,C 180,E1 12784.727,E2 12784.727} C_VEL
LIN {X 0,Y 348.499,Z 857.28,A -85,B 0,C 180,E1 12792.573,E2 12792.573} C_VEL
LIN {X 0,Y 348.266,Z 857.28,A -85,B 0,C 180,E1 12797.743,E2 12797.743} C_VEL
LIN {X 0,Y 347.865,Z 857.28,A -85,B 0,C 180,E1 12805.825,E2 12805.825} C_VEL
LIN {X 0,Y 347.654,Z 857.28,A -85,B 0,C 180,E1 12811.53,E2 12811.53} C_VEL
LIN {X 0,Y 347.412,Z 857.28,A -85,B 0,C 180,E1 12818.33,E2 12818.33} C_VEL
LIN {X 0,Y 347.4,Z 857.28,A -85,B 0,C 180,E1 12825.788,E2 12825.788} C_VEL
LIN {X 0,Y 347.711,Z 857.743,A -85,B 0,C 180,E1 12833.442,E2 12833.442} C_VEL
LIN {X 0,Y 370.597,Z 919.089,A -85,B 0,C 180,E1 12836.733,E2 12836.733} C_VEL
LIN {X 0,Y 368.109,Z 953.13,A -85,B 0,C 180,E1 12838.198,E2 12838.198} C_VEL
LIN {X 0,Y 364.006,Z 984.591,A -85,B 0,C 180,E1 12840.429,E2 12840.429} C_VEL
LIN {X 0,Y 359.504,Z 1014.186,A -85,B 0,C 180,E1 12843.587,E2 12843.587} C_VEL
LIN {X 0,Y 355.454,Z 1039.732,A -85,B 0,C 180,E1 12847.459,E2 12847.459} C_VEL
LIN {X 0,Y 352.431,Z 1061.125,A -85,B 0,C 180,E1 12852.014,E2 12852.014} C_VEL
LIN {X 0,Y 350.85,Z 1077.741,A -85,B 0,C 180,E1 12857.124,E2 12857.124} C_VEL
LIN {X 0,Y 350.546,Z 1088.925,A -85,B 0,C 180,E1 12862.556,E2 12862.556} C_VEL
LIN {X 0,Y 350.572,Z 1093.814,A -85,B 0,C 180,E1 12867.526,E2 12867.526} C_VEL
LIN {X 0,Y 350.743,Z 1094.494,A -85,B 0,C 180,E1 12870.001,E2 12870.001} C_VEL
LIN {X 0,Y 350.592,Z 1092.2,A -85,B 0,C 180,E1 12874.956,E2 12874.956} C_VEL
LIN {X 0,Y 350.549,Z 1083.769,A -85,B 0,C 180,E1 12880.578,E2 12880.578} C_VEL
LIN {X 0,Y 351.639,Z 1069.304,A -85,B 0,C 180,E1 12886.086,E2 12886.086} C_VEL
LIN {X 0,Y 350.899,Z 1065.12,A -85,B 0,C 180,E1 12887.334,E2 12887.334} C_VEL
LIN {X 0,Y 346.124,Z 1052.648,A -85,B 0,C 180,E1 12890.667,E2 12890.667} C_VEL
LIN {X 0,Y 346.266,Z 1051.358,A -85,B 0,C 180,E1 12890.963,E2 12890.963} C_VEL
LIN {X 0,Y 350.67,Z 1027.294,A -85,B 0,C 180,E1 12895.581,E2 12895.581} C_VEL
LIN {X 0,Y 356.105,Z 999.072,A -85,B 0,C 180,E1 12899.384,E2 12899.384} C_VEL
LIN {X 0,Y 361.587,Z 967.353,A -85,B 0,C 180,E1 12902.269,E2 12902.269} C_VEL
LIN {X 0,Y 365.892,Z 935.005,A -85,B 0,C 180,E1 12904.129,E2 12904.129} C_VEL
LIN {X 0,Y 366.511,Z 920.921,A -85,B 0,C 180,E1 12904.741,E2 12904.741} C_VEL
LIN {X 0,Y 356.591,Z 892.161,A -85,B 0,C 180,E1 12906.715,E2 12906.715} C_VEL
LIN {X 0,Y 339.535,Z 857.28,A -85,B 0,C 180,E1 12909.985,E2 12909.985} C_VEL
LIN {X 0,Y 339.471,Z 857.28,A -85,B 0,C 180,E1 12917.987,E2 12917.987} C_VEL
LIN {X 0,Y 339.526,Z 857.28,A -85,B 0,C 180,E1 12924.547,E2 12924.547} C_VEL
LIN {X 0,Y 339.784,Z 857.28,A -85,B 0,C 180,E1 12930.625,E2 12930.625} C_VEL
LIN {X 0,Y 340.143,Z 857.28,A -85,B 0,C 180,E1 12939.113,E2 12939.113} C_VEL
LIN {X 0,Y 340.428,Z 857.28,A -85,B 0,C 180,E1 12947.123,E2 12947.123} C_VEL
LIN {X 0,Y 341.029,Z 857.28,A -85,B 0,C 180,E1 12954.875,E2 12954.875} C_VEL
LIN {X 0,Y 341.378,Z 857.28,A -85,B 0,C 180,E1 12959.967,E2 12959.967} C_VEL
LIN {X 0,Y 340.852,Z 857.28,A -85,B 0,C 180,E1 12967.622,E2 12967.622} C_VEL
LIN {X 0,Y 340.455,Z 857.28,A -85,B 0,C 180,E1 12975.435,E2 12975.435} C_VEL
LIN {X 0,Y 340.003,Z 857.28,A -85,B 0,C 180,E1 12983.581,E2 12983.581} C_VEL
LIN {X 0,Y 339.772,Z 857.28,A -85,B 0,C 180,E1 12989.301,E2 12989.301} C_VEL
LIN {X 0,Y 339.449,Z 857.28,A -85,B 0,C 180,E1 12996.593,E2 12996.593} C_VEL
LIN {X 0,Y 339.478,Z 857.352,A -85,B 0,C 180,E1 13001.34,E2 13001.34} C_VEL
LIN {X 0,Y 345.844,Z 871.357,A -85,B 0,C 180,E1 13002.912,E2 13002.912} C_VEL
LIN {X 0,Y 355.544,Z 896.951,A -85,B 0,C 180,E1 13006.089,E2 13006.089} C_VEL
LIN {X 0,Y 360.286,Z 918.931,A -85,B 0,C 180,E1 13009.075,E2 13009.075} C_VEL
LIN {X 0,Y 356.041,Z 943.118,A -85,B 0,C 180,E1 13012.399,E2 13012.399} C_VEL
LIN {X 0,Y 351.554,Z 962.34,A -85,B 0,C 180,E1 13016.274,E2 13016.274} C_VEL
LIN {X 0,Y 347.734,Z 977.138,A -85,B 0,C 180,E1 13020.847,E2 13020.847} C_VEL
LIN {X 0,Y 345.389,Z 985.873,A -85,B 0,C 180,E1 13025.388,E2 13025.388} C_VEL
LIN {X 0,Y 344.153,Z 989.652,A -85,B 0,C 180,E1 13029.392,E2 13029.392} C_VEL
LIN {X 0,Y 343.677,Z 989.52,A -85,B 0,C 180,E1 13034.672,E2 13034.672} C_VEL
LIN {X 0,Y 344.678,Z 983.586,A -85,B 0,C 180,E1 13039.879,E2 13039.879} C_VEL
LIN {X 0,Y 346.414,Z 973.356,A -85,B 0,C 180,E1 13044.355,E2 13044.355} C_VEL
LIN {X 0,Y 349.068,Z 957.356,A -85,B 0,C 180,E1 13048.756,E2 13048.756} C_VEL
LIN {X 0,Y 352.715,Z 936.095,A -85,B 0,C 180,E1 13052.613,E2 13052.613} C_VEL
LIN {X 0,Y 355.445,Z 913.228,A -85,B 0,C 180,E1 13055.499,E2 13055.499} C_VEL
LIN {X 0,Y 350.542,Z 887.975,A -85,B 0,C 180,E1 13058.257,E2 13058.257} C_VEL
LIN {X 0,Y 341.178,Z 860,A -85,B 0,C 180,E1 13060.693,E2 13060.693} C_VEL
LIN {X 0,Y 340.663,Z 857.28,A -85,B 0,C 180,E1 13060.906,E2 13060.906} C_VEL
LIN {X 0,Y 340.266,Z 857.28,A -85,B 0,C 180,E1 13068.147,E2 13068.147} C_VEL
LIN {X 0,Y 339.77,Z 857.28,A -85,B 0,C 180,E1 13076.462,E2 13076.462} C_VEL
LIN {X 0,Y 339.618,Z 857.28,A -85,B 0,C 180,E1 13082.342,E2 13082.342} C_VEL
LIN {X 0,Y 339.444,Z 857.28,A -85,B 0,C 180,E1 13088.642,E2 13088.642} C_VEL
LIN {X 0,Y 339.699,Z 857.28,A -85,B 0,C 180,E1 13093.001,E2 13093.001} C_VEL
LIN {X 0,Y 348,Z 888.315,A -85,B 0,C 180,E1 13094.985,E2 13094.985} C_VEL
LIN {X 0,Y 351.858,Z 911.244,A -85,B 0,C 180,E1 13097.064,E2 13097.064} C_VEL
LIN {X 0,Y 349.387,Z 937.32,A -85,B 0,C 180,E1 13100.075,E2 13100.075} C_VEL
LIN {X 0,Y 347.057,Z 958.282,A -85,B 0,C 180,E1 13103.72,E2 13103.72} C_VEL
LIN {X 0,Y 345.378,Z 973.962,A -85,B 0,C 180,E1 13107.793,E2 13107.793} C_VEL
LIN {X 0,Y 344.244,Z 984.512,A -85,B 0,C 180,E1 13112.168,E2 13112.168} C_VEL
LIN {X 0,Y 343.761,Z 989.975,A -85,B 0,C 180,E1 13116.693,E2 13116.693} C_VEL
LIN {X 0,Y 343.901,Z 990.839,A -85,B 0,C 180,E1 13119.421,E2 13119.421} C_VEL
LIN {X 0,Y 344.749,Z 988.718,A -85,B 0,C 180,E1 13123.454,E2 13123.454} C_VEL
LIN {X 0,Y 346.508,Z 981.044,A -85,B 0,C 180,E1 13128.104,E2 13128.104} C_VEL
LIN {X 0,Y 349.165,Z 967.336,A -85,B 0,C 180,E1 13132.561,E2 13132.561} C_VEL
LIN {X 0,Y 352.302,Z 948.919,A -85,B 0,C 180,E1 13136.337,E2 13136.337} C_VEL
LIN {X 0,Y 355.296,Z 926.266,A -85,B 0,C 180,E1 13139.421,E2 13139.421} C_VEL
LIN {X 0,Y 356.348,Z 908.102,A -85,B 0,C 180,E1 13141.216,E2 13141.216} C_VEL
LIN {X 0,Y 351.225,Z 883.251,A -85,B 0,C 180,E1 13143.499,E2 13143.499} C_VEL
LIN {X 0,Y 340.956,Z 857.28,A -85,B 0,C 180,E1 13145.765,E2 13145.765} C_VEL
LIN {X 0,Y 340.542,Z 857.28,A -85,B 0,C 180,E1 13152.872,E2 13152.872} C_VEL
LIN {X 0,Y 340.137,Z 857.28,A -85,B 0,C 180,E1 13160.887,E2 13160.887} C_VEL
LIN {X 0,Y 339.786,Z 857.28,A -85,B 0,C 180,E1 13169.374,E2 13169.374} C_VEL
LIN {X 0,Y 339.463,Z 857.28,A -85,B 0,C 180,E1 13176.599,E2 13176.599} C_VEL
LIN {X 0,Y 339.5,Z 857.28,A -85,B 0,C 180,E1 13184.476,E2 13184.476} C_VEL
LIN {X 0,Y 339.667,Z 857.28,A -85,B 0,C 180,E1 13192.637,E2 13192.637} C_VEL
LIN {X 0,Y 362.982,Z 919.303,A -85,B 0,C 180,E1 13196.173,E2 13196.173} C_VEL
LIN {X 0,Y 362.759,Z 934.238,A -85,B 0,C 180,E1 13196.777,E2 13196.777} C_VEL
LIN {X 0,Y 358.784,Z 968.489,A -85,B 0,C 180,E1 13198.696,E2 13198.696} C_VEL
LIN {X 0,Y 354.308,Z 999.392,A -85,B 0,C 180,E1 13201.482,E2 13201.482} C_VEL
LIN {X 0,Y 349.544,Z 1027.944,A -85,B 0,C 180,E1 13205.249,E2 13205.249} C_VEL
LIN {X 0,Y 345.869,Z 1050.779,A -85,B 0,C 180,E1 13209.501,E2 13209.501} C_VEL
LIN {X 0,Y 343.476,Z 1070.259,A -85,B 0,C 180,E1 13214.665,E2 13214.665} C_VEL
LIN {X 0,Y 342.706,Z 1083.192,A -85,B 0,C 180,E1 13219.822,E2 13219.822} C_VEL
LIN {X 0,Y 342.766,Z 1090.735,A -85,B 0,C 180,E1 13224.933,E2 13224.933} C_VEL
LIN {X 0,Y 342.927,Z 1093.309,A -85,B 0,C 180,E1 13230.001,E2 13230.001} C_VEL
LIN {X 0,Y 342.757,Z 1091.049,A -85,B 0,C 180,E1 13235.069,E2 13235.069} C_VEL
LIN {X 0,Y 342.696,Z 1082.632,A -85,B 0,C 180,E1 13240.824,E2 13240.824} C_VEL
LIN {X 0,Y 343.818,Z 1068.692,A -85,B 0,C 180,E1 13246.305,E2 13246.305} C_VEL
LIN {X 0,Y 346.266,Z 1051.358,A -85,B 0,C 180,E1 13250.963,E2 13250.963} C_VEL
LIN {X 0,Y 344.36,Z 1041.09,A -85,B 0,C 180,E1 13253.298,E2 13253.298} C_VEL
LIN {X 0,Y 342.652,Z 1029.955,A -85,B 0,C 180,E1 13255.548,E2 13255.548} C_VEL
LIN {X 0,Y 348.07,Z 1003.39,A -85,B 0,C 180,E1 13259.405,E2 13259.405} C_VEL
LIN {X 0,Y 353.568,Z 974.16,A -85,B 0,C 180,E1 13262.364,E2 13262.364} C_VEL
LIN {X 0,Y 358.457,Z 941.482,A -85,B 0,C 180,E1 13264.503,E2 13264.503} C_VEL
LIN {X 0,Y 359.805,Z 922.815,A -85,B 0,C 180,E1 13265.364,E2 13265.364} C_VEL
LIN {X 0,Y 350.375,Z 895.149,A -85,B 0,C 180,E1 13267.397,E2 13267.397} C_VEL
LIN {X 0,Y 333.642,Z 862.586,A -85,B 0,C 180,E1 13270.547,E2 13270.547} C_VEL
LIN {X 0,Y 331.551,Z 857.28,A -85,B 0,C 180,E1 13271.114,E2 13271.114} C_VEL
LIN {X 0,Y 331.514,Z 857.28,A -85,B 0,C 180,E1 13276.95,E2 13276.95} C_VEL
LIN {X 0,Y 331.605,Z 857.28,A -85,B 0,C 180,E1 13283.566,E2 13283.566} C_VEL
LIN {X 0,Y 331.818,Z 857.28,A -85,B 0,C 180,E1 13290.11,E2 13290.11} C_VEL
LIN {X 0,Y 332.153,Z 857.28,A -85,B 0,C 180,E1 13298.587,E2 13298.587} C_VEL
LIN {X 0,Y 332.368,Z 857.28,A -85,B 0,C 180,E1 13304.11,E2 13304.11} C_VEL
LIN {X 0,Y 332.931,Z 857.28,A -85,B 0,C 180,E1 13312.128,E2 13312.128} C_VEL
LIN {X 0,Y 333.475,Z 857.28,A -85,B 0,C 180,E1 13319.967,E2 13319.967} C_VEL
LIN {X 0,Y 332.922,Z 857.28,A -85,B 0,C 180,E1 13327.805,E2 13327.805} C_VEL
LIN {X 0,Y 332.486,Z 857.28,A -85,B 0,C 180,E1 13335.815,E2 13335.815} C_VEL
LIN {X 0,Y 332.015,Z 857.28,A -85,B 0,C 180,E1 13344.184,E2 13344.184} C_VEL
LIN {X 0,Y 331.78,Z 857.28,A -85,B 0,C 180,E1 13350.078,E2 13350.078} C_VEL
LIN {X 0,Y 331.563,Z 857.28,A -85,B 0,C 180,E1 13356.356,E2 13356.356} C_VEL
LIN {X 0,Y 331.541,Z 857.64,A -85,B 0,C 180,E1 13360.153,E2 13360.153} C_VEL
LIN {X 0,Y 344.508,Z 886.251,A -85,B 0,C 180,E1 13363.736,E2 13363.736} C_VEL
LIN {X 0,Y 351.902,Z 912.118,A -85,B 0,C 180,E1 13367.231,E2 13367.231} C_VEL
LIN {X 0,Y 353.074,Z 925.217,A -85,B 0,C 180,E1 13369.093,E2 13369.093} C_VEL
LIN {X 0,Y 348.188,Z 948.083,A -85,B 0,C 180,E1 13372.497,E2 13372.497} C_VEL
LIN {X 0,Y 343.459,Z 966.759,A -85,B 0,C 180,E1 13376.642,E2 13376.642} C_VEL
LIN {X 0,Y 339.663,Z 980.422,A -85,B 0,C 180,E1 13381.367,E2 13381.367} C_VEL
LIN {X 0,Y 337.319,Z 988.365,A -85,B 0,C 180,E1 13386.172,E2 13386.172} C_VEL
LIN {X 0,Y 335.949,Z 991.473,A -85,B 0,C 180,E1 13391.609,E2 13391.609} C_VEL
LIN {X 0,Y 336.127,Z 988.804,A -85,B 0,C 180,E1 13396.983,E2 13396.983} C_VEL
LIN {X 0,Y 337.675,Z 980.289,A -85,B 0,C 180,E1 13402.269,E2 13402.269} C_VEL
LIN {X 0,Y 340.05,Z 966.238,A -85,B 0,C 180,E1 13407.128,E2 13407.128} C_VEL
LIN {X 0,Y 343.434,Z 947.713,A -85,B 0,C 180,E1 13411.262,E2 13411.262} C_VEL
LIN {X 0,Y 347.359,Z 923.803,A -85,B 0,C 180,E1 13414.844,E2 13414.844} C_VEL
LIN {X 0,Y 347.688,Z 912.196,A -85,B 0,C 180,E1 13416.24,E2 13416.24} C_VEL
LIN {X 0,Y 342.765,Z 887.817,A -85,B 0,C 180,E1 13418.938,E2 13418.938} C_VEL
LIN {X 0,Y 333.319,Z 860.096,A -85,B 0,C 180,E1 13421.417,E2 13421.417} C_VEL
LIN {X 0,Y 332.774,Z 857.28,A -85,B 0,C 180,E1 13421.769,E2 13421.769} C_VEL
LIN {X 0,Y 332.299,Z 857.28,A -85,B 0,C 180,E1 13428.598,E2 13428.598} C_VEL
LIN {X 0,Y 331.823,Z 857.28,A -85,B 0,C 180,E1 13437.147,E2 13437.147} C_VEL
LIN {X 0,Y 331.521,Z 857.28,A -85,B 0,C 180,E1 13444.802,E2 13444.802} C_VEL
LIN {X 0,Y 331.755,Z 857.971,A -85,B 0,C 180,E1 13452.565,E2 13452.565} C_VEL
LIN {X 0,Y 339.866,Z 887.095,A -85,B 0,C 180,E1 13454.403,E2 13454.403} C_VEL
LIN {X 0,Y 344.447,Z 911.117,A -85,B 0,C 180,E1 13456.601,E2 13456.601} C_VEL
LIN {X 0,Y 341.904,Z 937.031,A -85,B 0,C 180,E1 13459.584,E2 13459.584} C_VEL
LIN {X 0,Y 339.605,Z 957.295,A -85,B 0,C 180,E1 13463.056,E2 13463.056} C_VEL
LIN {X 0,Y 337.651,Z 974.596,A -85,B 0,C 180,E1 13467.501,E2 13467.501} C_VEL
LIN {X 0,Y 336.445,Z 985.724,A -85,B 0,C 180,E1 13472.153,E2 13472.153} C_VEL
LIN {X 0,Y 335.969,Z 990.751,A -85,B 0,C 180,E1 13476.119,E2 13476.119} C_VEL
LIN {X 0,Y 336.361,Z 991.849,A -85,B 0,C 180,E1 13480.956,E2 13480.956} C_VEL
LIN {X 0,Y 337.818,Z 987.165,A -85,B 0,C 180,E1 13485.89,E2 13485.89} C_VEL
LIN {X 0,Y 340.063,Z 977.228,A -85,B 0,C 180,E1 13490.426,E2 13490.426} C_VEL
LIN {X 0,Y 343.161,Z 961.452,A -85,B 0,C 180,E1 13494.687,E2 13494.687} C_VEL
LIN {X 0,Y 346.647,Z 940.263,A -85,B 0,C 180,E1 13498.39,E2 13498.39} C_VEL
LIN {X 0,Y 349.732,Z 915.578,A -85,B 0,C 180,E1 13501.19,E2 13501.19} C_VEL
LIN {X 0,Y 346.117,Z 891.084,A -85,B 0,C 180,E1 13503.605,E2 13503.605} C_VEL
LIN {X 0,Y 337.206,Z 866.997,A -85,B 0,C 180,E1 13505.803,E2 13505.803} C_VEL
LIN {X 0,Y 332.951,Z 857.28,A -85,B 0,C 180,E1 13506.837,E2 13506.837} C_VEL
LIN {X 0,Y 332.586,Z 857.28,A -85,B 0,C 180,E1 13513.186,E2 13513.186} C_VEL
LIN {X 0,Y 332.315,Z 857.28,A -85,B 0,C 180,E1 13518.625,E2 13518.625} C_VEL
LIN {X 0,Y 332.019,Z 857.28,A -85,B 0,C 180,E1 13524.257,E2 13524.257} C_VEL
LIN {X 0,Y 331.788,Z 857.28,A -85,B 0,C 180,E1 13530.155,E2 13530.155} C_VEL
LIN {X 0,Y 331.587,Z 857.28,A -85,B 0,C 180,E1 13536.436,E2 13536.436} C_VEL
LIN {X 0,Y 331.52,Z 857.28,A -85,B 0,C 180,E1 13543.263,E2 13543.263} C_VEL
LIN {X 0,Y 331.617,Z 857.28,A -85,B 0,C 180,E1 13550.934,E2 13550.934} C_VEL
LIN {X 0,Y 331.687,Z 857.28,A -85,B 0,C 180,E1 13551.923,E2 13551.923} C_VEL
LIN {X 0,Y 354.4,Z 916.836,A -85,B 0,C 180,E1 13555.422,E2 13555.422} C_VEL
LIN {X 0,Y 356.343,Z 925.29,A -85,B 0,C 180,E1 13555.898,E2 13555.898} C_VEL
LIN {X 0,Y 352.739,Z 959.204,A -85,B 0,C 180,E1 13557.582,E2 13557.582} C_VEL
LIN {X 0,Y 348.158,Z 990.898,A -85,B 0,C 180,E1 13560.186,E2 13560.186} C_VEL
LIN {X 0,Y 343.361,Z 1019.373,A -85,B 0,C 180,E1 13563.66,E2 13563.66} C_VEL
LIN {X 0,Y 339.051,Z 1044.549,A -85,B 0,C 180,E1 13568.039,E2 13568.039} C_VEL
LIN {X 0,Y 336.331,Z 1064.596,A -85,B 0,C 180,E1 13572.986,E2 13572.986} C_VEL
LIN {X 0,Y 334.954,Z 1079.122,A -85,B 0,C 180,E1 13578.264,E2 13578.264} C_VEL
LIN {X 0,Y 334.903,Z 1088,A -85,B 0,C 180,E1 13583.445,E2 13583.445} C_VEL
LIN {X 0,Y 334.934,Z 1091.411,A -85,B 0,C 180,E1 13587.41,E2 13587.41} C_VEL
LIN {X 0,Y 335.111,Z 1092.121,A -85,B 0,C 180,E1 13590.001,E2 13590.001} C_VEL
LIN {X 0,Y 334.858,Z 1089.278,A -85,B 0,C 180,E1 13595.796,E2 13595.796} C_VEL
LIN {X 0,Y 334.844,Z 1081.505,A -85,B 0,C 180,E1 13601.081,E2 13601.081} C_VEL
LIN {X 0,Y 336.144,Z 1067.613,A -85,B 0,C 180,E1 13606.688,E2 13606.688} C_VEL
LIN {X 0,Y 339.159,Z 1048.148,A -85,B 0,C 180,E1 13611.956,E2 13611.956} C_VEL
LIN {X 0,Y 342.652,Z 1029.955,A -85,B 0,C 180,E1 13615.548,E2 13615.548} C_VEL
LIN {X 0,Y 341.384,Z 1018.122,A -85,B 0,C 180,E1 13617.716,E2 13617.716} C_VEL
LIN {X 0,Y 340.478,Z 1005.336,A -85,B 0,C 180,E1 13619.721,E2 13619.721} C_VEL
LIN {X 0,Y 346.512,Z 975.061,A -85,B 0,C 180,E1 13622.92,E2 13622.92} C_VEL
LIN {X 0,Y 351.637,Z 942.884,A -85,B 0,C 180,E1 13625.128,E2 13625.128} C_VEL
LIN {X 0,Y 353.091,Z 924.473,A -85,B 0,C 180,E1 13626.033,E2 13626.033} C_VEL
LIN {X 0,Y 343.838,Z 897.164,A -85,B 0,C 180,E1 13628.182,E2 13628.182} C_VEL
LIN {X 0,Y 328.101,Z 866.919,A -85,B 0,C 180,E1 13631.275,E2 13631.275} C_VEL
LIN {X 0,Y 323.69,Z 858.168,A -85,B 0,C 180,E1 13632.24,E2 13632.24} C_VEL
LIN {X 0,Y 323.621,Z 857.28,A -85,B 0,C 180,E1 13632.388,E2 13632.388} C_VEL
LIN {X 0,Y 323.518,Z 857.28,A -85,B 0,C 180,E1 13639.041,E2 13639.041} C_VEL
LIN {X 0,Y 323.684,Z 857.28,A -85,B 0,C 180,E1 13645.829,E2 13645.829} C_VEL
LIN {X 0,Y 323.994,Z 857.28,A -85,B 0,C 180,E1 13652.613,E2 13652.613} C_VEL
LIN {X 0,Y 324.317,Z 857.28,A -85,B 0,C 180,E1 13660.898,E2 13660.898} C_VEL
LIN {X 0,Y 324.701,Z 857.28,A -85,B 0,C 180,E1 13669.22,E2 13669.22} C_VEL
LIN {X 0,Y 325.447,Z 857.28,A -85,B 0,C 180,E1 13677.3,E2 13677.3} C_VEL
LIN {X 0,Y 325.43,Z 857.28,A -85,B 0,C 180,E1 13682.631,E2 13682.631} C_VEL
LIN {X 0,Y 324.79,Z 857.28,A -85,B 0,C 180,E1 13690.707,E2 13690.707} C_VEL
LIN {X 0,Y 324.539,Z 857.28,A -85,B 0,C 180,E1 13696.213,E2 13696.213} C_VEL
LIN {X 0,Y 324.188,Z 857.28,A -85,B 0,C 180,E1 13701.893,E2 13701.893} C_VEL
LIN {X 0,Y 323.897,Z 857.28,A -85,B 0,C 180,E1 13707.817,E2 13707.817} C_VEL
LIN {X 0,Y 323.664,Z 857.28,A -85,B 0,C 180,E1 13714.091,E2 13714.091} C_VEL
LIN {X 0,Y 323.607,Z 857.28,A -85,B 0,C 180,E1 13718.829,E2 13718.829} C_VEL
LIN {X 0,Y 327.732,Z 866.719,A -85,B 0,C 180,E1 13719.962,E2 13719.962} C_VEL
LIN {X 0,Y 338.414,Z 890.278,A -85,B 0,C 180,E1 13723.224,E2 13723.224} C_VEL
LIN {X 0,Y 345.079,Z 914.754,A -85,B 0,C 180,E1 13726.7,E2 13726.7} C_VEL
LIN {X 0,Y 346.326,Z 926.42,A -85,B 0,C 180,E1 13728.452,E2 13728.452} C_VEL
LIN {X 0,Y 341.229,Z 949.079,A -85,B 0,C 180,E1 13731.883,E2 13731.883} C_VEL
LIN {X 0,Y 336.269,Z 967.609,A -85,B 0,C 180,E1 13736.057,E2 13736.057} C_VEL
LIN {X 0,Y 332.333,Z 980.936,A -85,B 0,C 180,E1 13740.674,E2 13740.674} C_VEL
LIN {X 0,Y 329.763,Z 989.219,A -85,B 0,C 180,E1 13745.591,E2 13745.591} C_VEL
LIN {X 0,Y 328.198,Z 992.643,A -85,B 0,C 180,E1 13751.159,E2 13751.159} C_VEL
LIN {X 0,Y 328.254,Z 990.298,A -85,B 0,C 180,E1 13756.665,E2 13756.665} C_VEL
LIN {X 0,Y 329.786,Z 982.14,A -85,B 0,C 180,E1 13762.082,E2 13762.082} C_VEL
LIN {X 0,Y 332.145,Z 968.601,A -85,B 0,C 180,E1 13767.059,E2 13767.059} C_VEL
LIN {X 0,Y 335.557,Z 950.679,A -85,B 0,C 180,E1 13771.292,E2 13771.292} C_VEL
LIN {X 0,Y 339.651,Z 927.602,A -85,B 0,C 180,E1 13774.954,E2 13774.954} C_VEL
LIN {X 0,Y 340.481,Z 914.863,A -85,B 0,C 180,E1 13776.542,E2 13776.542} C_VEL
LIN {X 0,Y 335.724,Z 890.407,A -85,B 0,C 180,E1 13779.377,E2 13779.377} C_VEL
LIN {X 0,Y 326.265,Z 861.751,A -85,B 0,C 180,E1 13782.039,E2 13782.039} C_VEL
LIN {X 0,Y 324.863,Z 857.28,A -85,B 0,C 180,E1 13782.493,E2 13782.493} C_VEL
LIN {X 0,Y 324.31,Z 857.28,A -85,B 0,C 180,E1 13789.074,E2 13789.074} C_VEL
LIN {X 0,Y 323.888,Z 857.28,A -85,B 0,C 180,E1 13797.475,E2 13797.475} C_VEL
LIN {X 0,Y 323.613,Z 857.28,A -85,B 0,C 180,E1 13804.154,E2 13804.154} C_VEL
LIN {X 0,Y 323.757,Z 857.28,A -85,B 0,C 180,E1 13811.985,E2 13811.985} C_VEL
LIN {X 0,Y 332.267,Z 888.189,A -85,B 0,C 180,E1 13813.992,E2 13813.992} C_VEL
LIN {X 0,Y 336.861,Z 912.881,A -85,B 0,C 180,E1 13816.312,E2 13816.312} C_VEL
LIN {X 0,Y 334.254,Z 938.263,A -85,B 0,C 180,E1 13819.311,E2 13819.311} C_VEL
LIN {X 0,Y 331.782,Z 959.411,A -85,B 0,C 180,E1 13823.054,E2 13823.054} C_VEL
LIN {X 0,Y 329.925,Z 975.158,A -85,B 0,C 180,E1 13827.186,E2 13827.186} C_VEL
LIN {X 0,Y 328.672,Z 986.382,A -85,B 0,C 180,E1 13831.819,E2 13831.819} C_VEL
LIN {X 0,Y 328.169,Z 991.406,A -85,B 0,C 180,E1 13835.514,E2 13835.514} C_VEL
LIN {X 0,Y 328.209,Z 993.152,A -85,B 0,C 180,E1 13838.389,E2 13838.389} C_VEL
LIN {X 0,Y 328.632,Z 993.072,A -85,B 0,C 180,E1 13841.23,E2 13841.23} C_VEL
LIN {X 0,Y 330.012,Z 989.126,A -85,B 0,C 180,E1 13845.756,E2 13845.756} C_VEL
LIN {X 0,Y 332.202,Z 980.242,A -85,B 0,C 180,E1 13850.197,E2 13850.197} C_VEL
LIN {X 0,Y 335.233,Z 966.006,A -85,B 0,C 180,E1 13854.444,E2 13854.444} C_VEL
LIN {X 0,Y 338.912,Z 946.107,A -85,B 0,C 180,E1 13858.273,E2 13858.273} C_VEL
LIN {X 0,Y 342.193,Z 923.039,A -85,B 0,C 180,E1 13861.216,E2 13861.216} C_VEL
LIN {X 0,Y 342.346,Z 909.998,A -85,B 0,C 180,E1 13862.566,E2 13862.566} C_VEL
LIN {X 0,Y 337.135,Z 885.38,A -85,B 0,C 180,E1 13865.02,E2 13865.02} C_VEL
LIN {X 0,Y 326.688,Z 862.085,A -85,B 0,C 180,E1 13867.406,E2 13867.406} C_VEL
LIN {X 0,Y 325.023,Z 857.28,A -85,B 0,C 180,E1 13867.86,E2 13867.86} C_VEL
LIN {X 0,Y 324.508,Z 857.28,A -85,B 0,C 180,E1 13876.285,E2 13876.285} C_VEL
LIN {X 0,Y 324.19,Z 857.28,A -85,B 0,C 180,E1 13881.966,E2 13881.966} C_VEL
LIN {X 0,Y 323.929,Z 857.28,A -85,B 0,C 180,E1 13887.892,E2 13887.892} C_VEL
LIN {X 0,Y 323.673,Z 857.28,A -85,B 0,C 180,E1 13894.173,E2 13894.173} C_VEL
LIN {X 0,Y 323.496,Z 857.28,A -85,B 0,C 180,E1 13901.51,E2 13901.51} C_VEL
LIN {X 0,Y 323.548,Z 857.28,A -85,B 0,C 180,E1 13909.071,E2 13909.071} C_VEL
LIN {X 0,Y 323.757,Z 857.28,A -85,B 0,C 180,E1 13911.085,E2 13911.085} C_VEL
LIN {X 0,Y 346.484,Z 916.215,A -85,B 0,C 180,E1 13914.758,E2 13914.758} C_VEL
LIN {X 0,Y 349.104,Z 927.114,A -85,B 0,C 180,E1 13915.408,E2 13915.408} C_VEL
LIN {X 0,Y 345.189,Z 961.294,A -85,B 0,C 180,E1 13917.22,E2 13917.22} C_VEL
LIN {X 0,Y 340.36,Z 993.016,A -85,B 0,C 180,E1 13919.986,E2 13919.986} C_VEL
LIN {X 0,Y 335.201,Z 1022.067,A -85,B 0,C 180,E1 13923.748,E2 13923.748} C_VEL
LIN {X 0,Y 330.725,Z 1047.492,A -85,B 0,C 180,E1 13928.517,E2 13928.517} C_VEL
LIN {X 0,Y 328.05,Z 1067.305,A -85,B 0,C 180,E1 13933.924,E2 13933.924} C_VEL
LIN {X 0,Y 327.024,Z 1080.519,A -85,B 0,C 180,E1 13939.328,E2 13939.328} C_VEL
LIN {X 0,Y 327.101,Z 1088.239,A -85,B 0,C 180,E1 13944.689,E2 13944.689} C_VEL
LIN {X 0,Y 327.304,Z 1090.934,A -85,B 0,C 180,E1 13950.001,E2 13950.001} C_VEL
LIN {X 0,Y 327.069,Z 1088.741,A -85,B 0,C 180,E1 13955.313,E2 13955.313} C_VEL
LIN {X 0,Y 326.93,Z 1081.65,A -85,B 0,C 180,E1 13960.677,E2 13960.677} C_VEL
LIN {X 0,Y 327.91,Z 1069.401,A -85,B 0,C 180,E1 13966.085,E2 13966.085} C_VEL
LIN {X 0,Y 330.752,Z 1051.297,A -85,B 0,C 180,E1 13971.483,E2 13971.483} C_VEL
LIN {X 0,Y 335.785,Z 1026.877,A -85,B 0,C 180,E1 13976.52,E2 13976.52} C_VEL
LIN {X 0,Y 340.478,Z 1005.336,A -85,B 0,C 180,E1 13979.721,E2 13979.721} C_VEL
LIN {X 0,Y 339.808,Z 991.882,A -85,B 0,C 180,E1 13981.617,E2 13981.617} C_VEL
LIN {X 0,Y 339.149,Z 977.719,A -85,B 0,C 180,E1 13983.349,E2 13983.349} C_VEL
LIN {X 0,Y 344.61,Z 946.005,A -85,B 0,C 180,E1 13985.691,E2 13985.691} C_VEL
LIN {X 0,Y 346.539,Z 926.353,A -85,B 0,C 180,E1 13986.71,E2 13986.71} C_VEL
LIN {X 0,Y 337.331,Z 899.228,A -85,B 0,C 180,E1 13989.003,E2 13989.003} C_VEL
LIN {X 0,Y 321.269,Z 868.34,A -85,B 0,C 180,E1 13992.338,E2 13992.338} C_VEL
LIN {X 0,Y 315.8,Z 858.789,A -85,B 0,C 180,E1 13993.582,E2 13993.582} C_VEL
LIN {X 0,Y 315.637,Z 857.28,A -85,B 0,C 180,E1 13993.756,E2 13993.756} C_VEL
LIN {X 0,Y 315.566,Z 857.28,A -85,B 0,C 180,E1 14001.385,E2 14001.385} C_VEL
LIN {X 0,Y 315.814,Z 857.28,A -85,B 0,C 180,E1 14009.652,E2 14009.652} C_VEL
LIN {X 0,Y 316.162,Z 857.28,A -85,B 0,C 180,E1 14017.446,E2 14017.446} C_VEL
LIN {X 0,Y 316.474,Z 857.28,A -85,B 0,C 180,E1 14023.289,E2 14023.289} C_VEL
LIN {X 0,Y 317.031,Z 857.28,A -85,B 0,C 180,E1 14031.731,E2 14031.731} C_VEL
LIN {X 0,Y 317.698,Z 857.28,A -85,B 0,C 180,E1 14039.965,E2 14039.965} C_VEL
LIN {X 0,Y 317.038,Z 857.28,A -85,B 0,C 180,E1 14048.198,E2 14048.198} C_VEL
LIN {X 0,Y 316.557,Z 857.28,A -85,B 0,C 180,E1 14056.633,E2 14056.633} C_VEL
LIN {X 0,Y 316.115,Z 857.28,A -85,B 0,C 180,E1 14064.488,E2 14064.488} C_VEL
LIN {X 0,Y 315.776,Z 857.28,A -85,B 0,C 180,E1 14071.775,E2 14071.775} C_VEL
LIN {X 0,Y 315.697,Z 857.28,A -85,B 0,C 180,E1 14077.441,E2 14077.441} C_VEL
LIN {X 0,Y 318.145,Z 863.003,A -85,B 0,C 180,E1 14078.156,E2 14078.156} C_VEL
LIN {X 0,Y 330.698,Z 889.868,A -85,B 0,C 180,E1 14082.04,E2 14082.04} C_VEL
LIN {X 0,Y 337.606,Z 913.561,A -85,B 0,C 180,E1 14085.549,E2 14085.549} C_VEL
LIN {X 0,Y 339.285,Z 929.144,A -85,B 0,C 180,E1 14087.979,E2 14087.979} C_VEL
LIN {X 0,Y 333.781,Z 952.064,A -85,B 0,C 180,E1 14091.625,E2 14091.625} C_VEL
LIN {X 0,Y 328.593,Z 970.18,A -85,B 0,C 180,E1 14095.94,E2 14095.94} C_VEL
LIN {X 0,Y 324.56,Z 982.986,A -85,B 0,C 180,E1 14100.67,E2 14100.67} C_VEL
LIN {X 0,Y 321.779,Z 991.241,A -85,B 0,C 180,E1 14106.117,E2 14106.117} C_VEL
LIN {X 0,Y 320.471,Z 993.816,A -85,B 0,C 180,E1 14110.716,E2 14110.716} C_VEL
LIN {X 0,Y 320.417,Z 991.788,A -85,B 0,C 180,E1 14116.333,E2 14116.333} C_VEL
LIN {X 0,Y 321.876,Z 983.986,A -85,B 0,C 180,E1 14121.887,E2 14121.887} C_VEL
LIN {X 0,Y 324.264,Z 970.86,A -85,B 0,C 180,E1 14126.988,E2 14126.988} C_VEL
LIN {X 0,Y 327.689,Z 953.495,A -85,B 0,C 180,E1 14131.323,E2 14131.323} C_VEL
LIN {X 0,Y 332.075,Z 930.119,A -85,B 0,C 180,E1 14135.231,E2 14135.231} C_VEL
LIN {X 0,Y 333.299,Z 917.561,A -85,B 0,C 180,E1 14136.848,E2 14136.848} C_VEL
LIN {X 0,Y 328.659,Z 892.891,A -85,B 0,C 180,E1 14139.827,E2 14139.827} C_VEL
LIN {X 0,Y 319.682,Z 865.391,A -85,B 0,C 180,E1 14142.538,E2 14142.538} C_VEL
LIN {X 0,Y 316.857,Z 857.28,A -85,B 0,C 180,E1 14143.206,E2 14143.206} C_VEL
LIN {X 0,Y 316.345,Z 857.28,A -85,B 0,C 180,E1 14149.573,E2 14149.573} C_VEL
LIN {X 0,Y 315.977,Z 857.28,A -85,B 0,C 180,E1 14155.546,E2 14155.546} C_VEL
LIN {X 0,Y 315.712,Z 857.28,A -85,B 0,C 180,E1 14161.838,E2 14161.838} C_VEL
LIN {X 0,Y 315.587,Z 857.28,A -85,B 0,C 180,E1 14169.944,E2 14169.944} C_VEL
LIN {X 0,Y 315.808,Z 857.515,A -85,B 0,C 180,E1 14171.49,E2 14171.49} C_VEL
LIN {X 0,Y 324.014,Z 886.574,A -85,B 0,C 180,E1 14173.339,E2 14173.339} C_VEL
LIN {X 0,Y 329.329,Z 912.898,A -85,B 0,C 180,E1 14175.836,E2 14175.836} C_VEL
LIN {X 0,Y 326.799,Z 938.088,A -85,B 0,C 180,E1 14178.828,E2 14178.828} C_VEL
LIN {X 0,Y 324.159,Z 959.821,A -85,B 0,C 180,E1 14182.675,E2 14182.675} C_VEL
LIN {X 0,Y 322.219,Z 975.818,A -85,B 0,C 180,E1 14186.895,E2 14186.895} C_VEL
LIN {X 0,Y 320.839,Z 987.758,A -85,B 0,C 180,E1 14191.894,E2 14191.894} C_VEL
LIN {X 0,Y 320.336,Z 993.565,A -85,B 0,C 180,E1 14196.752,E2 14196.752} C_VEL
LIN {X 0,Y 320.743,Z 994.511,A -85,B 0,C 180,E1 14200.75,E2 14200.75} C_VEL
LIN {X 0,Y 322.164,Z 991.116,A -85,B 0,C 180,E1 14205.514,E2 14205.514} C_VEL
LIN {X 0,Y 324.772,Z 981.474,A -85,B 0,C 180,E1 14210.648,E2 14210.648} C_VEL
LIN {X 0,Y 328.122,Z 966.808,A -85,B 0,C 180,E1 14215.073,E2 14215.073} C_VEL
LIN {X 0,Y 331.932,Z 947.474,A -85,B 0,C 180,E1 14218.858,E2 14218.858} C_VEL
LIN {X 0,Y 335.548,Z 923.258,A -85,B 0,C 180,E1 14221.972,E2 14221.972} C_VEL
LIN {X 0,Y 335.124,Z 908.007,A -85,B 0,C 180,E1 14223.624,E2 14223.624} C_VEL
LIN {X 0,Y 329.49,Z 884.637,A -85,B 0,C 180,E1 14226.056,E2 14226.056} C_VEL
LIN {X 0,Y 318.596,Z 862.076,A -85,B 0,C 180,E1 14228.643,E2 14228.643} C_VEL
LIN {X 0,Y 316.896,Z 857.28,A -85,B 0,C 180,E1 14229.311,E2 14229.311} C_VEL
LIN {X 0,Y 316.509,Z 857.28,A -85,B 0,C 180,E1 14236.919,E2 14236.919} C_VEL
LIN {X 0,Y 316.082,Z 857.28,A -85,B 0,C 180,E1 14245.565,E2 14245.565} C_VEL
LIN {X 0,Y 315.781,Z 857.28,A -85,B 0,C 180,E1 14251.857,E2 14251.857} C_VEL
LIN {X 0,Y 315.532,Z 857.28,A -85,B 0,C 180,E1 14259.849,E2 14259.849} C_VEL
LIN {X 0,Y 315.55,Z 857.28,A -85,B 0,C 180,E1 14267.799,E2 14267.799} C_VEL
LIN {X 0,Y 315.838,Z 857.899,A -85,B 0,C 180,E1 14270.336,E2 14270.336} C_VEL
LIN {X 0,Y 337.241,Z 911.747,A -85,B 0,C 180,E1 14273.806,E2 14273.806} C_VEL
LIN {X 0,Y 341.867,Z 929.244,A -85,B 0,C 180,E1 14274.92,E2 14274.92} C_VEL
LIN {X 0,Y 337.656,Z 963.199,A -85,B 0,C 180,E1 14276.837,E2 14276.837} C_VEL
LIN {X 0,Y 332.569,Z 994.885,A -85,B 0,C 180,E1 14279.76,E2 14279.76} C_VEL
LIN {X 0,Y 327.359,Z 1022.836,A -85,B 0,C 180,E1 14283.567,E2 14283.567} C_VEL
LIN {X 0,Y 322.943,Z 1047.116,A -85,B 0,C 180,E1 14288.301,E2 14288.301} C_VEL
LIN {X 0,Y 320.191,Z 1066.846,A -85,B 0,C 180,E1 14293.871,E2 14293.871} C_VEL
LIN {X 0,Y 319.179,Z 1080.422,A -85,B 0,C 180,E1 14299.754,E2 14299.754} C_VEL
LIN {X 0,Y 319.244,Z 1087.363,A -85,B 0,C 180,E1 14304.965,E2 14304.965} C_VEL
LIN {X 0,Y 319.488,Z 1089.744,A -85,B 0,C 180,E1 14310.001,E2 14310.001} C_VEL
LIN {X 0,Y 319.246,Z 1087.593,A -85,B 0,C 180,E1 14315.444,E2 14315.444} C_VEL
LIN {X 0,Y 319.07,Z 1080.539,A -85,B 0,C 180,E1 14320.943,E2 14320.943} C_VEL
LIN {X 0,Y 320.48,Z 1066.468,A -85,B 0,C 180,E1 14327.175,E2 14327.175} C_VEL
LIN {X 0,Y 323.859,Z 1047.5,A -85,B 0,C 180,E1 14332.688,E2 14332.688} C_VEL
LIN {X 0,Y 328.881,Z 1024.407,A -85,B 0,C 180,E1 14337.412,E2 14337.412} C_VEL
LIN {X 0,Y 335.148,Z 996.943,A -85,B 0,C 180,E1 14341.343,E2 14341.343} C_VEL
LIN {X 0,Y 339.149,Z 977.719,A -85,B 0,C 180,E1 14343.349,E2 14343.349} C_VEL
LIN {X 0,Y 338.653,Z 962.886,A -85,B 0,C 180,E1 14344.932,E2 14344.932} C_VEL
LIN {X 0,Y 337.841,Z 947.539,A -85,B 0,C 180,E1 14346.344,E2 14346.344} C_VEL
LIN {X 0,Y 339.932,Z 928.059,A -85,B 0,C 180,E1 14347.417,E2 14347.417} C_VEL
LIN {X 0,Y 331.053,Z 901.691,A -85,B 0,C 180,E1 14349.815,E2 14349.815} C_VEL
LIN {X 0,Y 316.183,Z 873.137,A -85,B 0,C 180,E1 14353.066,E2 14353.066} C_VEL
LIN {X 0,Y 307.739,Z 858.67,A -85,B 0,C 180,E1 14355.092,E2 14355.092} C_VEL
LIN {X 0,Y 307.59,Z 857.28,A -85,B 0,C 180,E1 14355.291,E2 14355.291} C_VEL
LIN {X 0,Y 307.622,Z 857.28,A -85,B 0,C 180,E1 14361.954,E2 14361.954} C_VEL
LIN {X 0,Y 307.924,Z 857.28,A -85,B 0,C 180,E1 14370.52,E2 14370.52} C_VEL
LIN {X 0,Y 308.266,Z 857.28,A -85,B 0,C 180,E1 14378.942,E2 14378.942} C_VEL
LIN {X 0,Y 308.612,Z 857.28,A -85,B 0,C 180,E1 14385.769,E2 14385.769} C_VEL
LIN {X 0,Y 309.323,Z 857.28,A -85,B 0,C 180,E1 14394.348,E2 14394.348} C_VEL
LIN {X 0,Y 309.794,Z 857.28,A -85,B 0,C 180,E1 14399.964,E2 14399.964} C_VEL
LIN {X 0,Y 309.096,Z 857.28,A -85,B 0,C 180,E1 14408.41,E2 14408.41} C_VEL
LIN {X 0,Y 308.603,Z 857.28,A -85,B 0,C 180,E1 14417.075,E2 14417.075} C_VEL
LIN {X 0,Y 308.225,Z 857.28,A -85,B 0,C 180,E1 14423.09,E2 14423.09} C_VEL
LIN {X 0,Y 307.911,Z 857.28,A -85,B 0,C 180,E1 14429.399,E2 14429.399} C_VEL
LIN {X 0,Y 307.698,Z 857.285,A -85,B 0,C 180,E1 14435.937,E2 14435.937} C_VEL
LIN {X 0,Y 310.012,Z 862.807,A -85,B 0,C 180,E1 14436.631,E2 14436.631} C_VEL
LIN {X 0,Y 322.508,Z 888.042,A -85,B 0,C 180,E1 14440.58,E2 14440.58} C_VEL
LIN {X 0,Y 329.959,Z 911.829,A -85,B 0,C 180,E1 14444.25,E2 14444.25} C_VEL
LIN {X 0,Y 332.649,Z 930.214,A -85,B 0,C 180,E1 14447.263,E2 14447.263} C_VEL
LIN {X 0,Y 327.062,Z 952.396,A -85,B 0,C 180,E1 14450.829,E2 14450.829} C_VEL
LIN {X 0,Y 321.674,Z 970.341,A -85,B 0,C 180,E1 14455.102,E2 14455.102} C_VEL
LIN {X 0,Y 317.178,Z 983.911,A -85,B 0,C 180,E1 14460.122,E2 14460.122} C_VEL
LIN {X 0,Y 314.247,Z 992.01,A -85,B 0,C 180,E1 14465.411,E2 14465.411} C_VEL
LIN {X 0,Y 312.751,Z 994.936,A -85,B 0,C 180,E1 14470.19,E2 14470.19} C_VEL
LIN {X 0,Y 312.566,Z 993.266,A -85,B 0,C 180,E1 14475.982,E2 14475.982} C_VEL
LIN {X 0,Y 313.987,Z 985.827,A -85,B 0,C 180,E1 14481.681,E2 14481.681} C_VEL
LIN {X 0,Y 316.413,Z 973.107,A -85,B 0,C 180,E1 14486.913,E2 14486.913} C_VEL
LIN {X 0,Y 320.165,Z 954.692,A -85,B 0,C 180,E1 14491.693,E2 14491.693} C_VEL
LIN {X 0,Y 324.73,Z 931.372,A -85,B 0,C 180,E1 14495.685,E2 14495.685} C_VEL
LIN {X 0,Y 325.888,Z 918.939,A -85,B 0,C 180,E1 14497.34,E2 14497.34} C_VEL
LIN {X 0,Y 321.65,Z 895.542,A -85,B 0,C 180,E1 14500.277,E2 14500.277} C_VEL
LIN {X 0,Y 312.798,Z 868.06,A -85,B 0,C 180,E1 14503.131,E2 14503.131} C_VEL
LIN {X 0,Y 308.789,Z 857.28,A -85,B 0,C 180,E1 14504.191,E2 14504.191} C_VEL
LIN {X 0,Y 308.223,Z 857.28,A -85,B 0,C 180,E1 14511.204,E2 14511.204} C_VEL
LIN {X 0,Y 307.843,Z 857.28,A -85,B 0,C 180,E1 14519.46,E2 14519.46} C_VEL
LIN {X 0,Y 307.598,Z 857.28,A -85,B 0,C 180,E1 14528.132,E2 14528.132} C_VEL
LIN {X 0,Y 307.837,Z 857.28,A -85,B 0,C 180,E1 14530.894,E2 14530.894} C_VEL
LIN {X 0,Y 316.821,Z 889.32,A -85,B 0,C 180,E1 14533.035,E2 14533.035} C_VEL
LIN {X 0,Y 321.786,Z 915.234,A -85,B 0,C 180,E1 14535.586,E2 14535.586} C_VEL
LIN {X 0,Y 318.982,Z 940.884,A -85,B 0,C 180,E1 14538.761,E2 14538.761} C_VEL
LIN {X 0,Y 316.181,Z 962.814,A -85,B 0,C 180,E1 14542.869,E2 14542.869} C_VEL
LIN {X 0,Y 314.177,Z 979.147,A -85,B 0,C 180,E1 14547.507,E2 14547.507} C_VEL
LIN {X 0,Y 312.953,Z 989.366,A -85,B 0,C 180,E1 14552.138,E2 14552.138} C_VEL
LIN {X 0,Y 312.525,Z 995.036,A -85,B 0,C 180,E1 14557.245,E2 14557.245} C_VEL
LIN {X 0,Y 312.855,Z 995.883,A -85,B 0,C 180,E1 14560.245,E2 14560.245} C_VEL
LIN {X 0,Y 314.078,Z 993.741,A -85,B 0,C 180,E1 14564.606,E2 14564.606} C_VEL
LIN {X 0,Y 316.464,Z 985.982,A -85,B 0,C 180,E1 14569.734,E2 14569.734} C_VEL
LIN {X 0,Y 320.038,Z 972.054,A -85,B 0,C 180,E1 14574.608,E2 14574.608} C_VEL
LIN {X 0,Y 324.127,Z 953.4,A -85,B 0,C 180,E1 14578.696,E2 14578.696} C_VEL
LIN {X 0,Y 328.087,Z 930.395,A -85,B 0,C 180,E1 14582.016,E2 14582.016} C_VEL
LIN {X 0,Y 329.058,Z 915.332,A -85,B 0,C 180,E1 14583.691,E2 14583.691} C_VEL
LIN {X 0,Y 324.568,Z 891.401,A -85,B 0,C 180,E1 14586.337,E2 14586.337} C_VEL
LIN {X 0,Y 314.29,Z 868.173,A -85,B 0,C 180,E1 14589.111,E2 14589.111} C_VEL
LIN {X 0,Y 308.988,Z 857.821,A -85,B 0,C 180,E1 14590.531,E2 14590.531} C_VEL
LIN {X 0,Y 308.586,Z 857.28,A -85,B 0,C 180,E1 14597.151,E2 14597.151} C_VEL
LIN {X 0,Y 308.224,Z 857.28,A -85,B 0,C 180,E1 14603.169,E2 14603.169} C_VEL
LIN {X 0,Y 307.92,Z 857.28,A -85,B 0,C 180,E1 14609.48,E2 14609.48} C_VEL
LIN {X 0,Y 307.61,Z 857.28,A -85,B 0,C 180,E1 14618.046,E2 14618.046} C_VEL
LIN {X 0,Y 307.61,Z 857.28,A -85,B 0,C 180,E1 14623.584,E2 14623.584} C_VEL
LIN {X 0,Y 307.754,Z 857.309,A -85,B 0,C 180,E1 14629.425,E2 14629.425} C_VEL
LIN {X 0,Y 329.419,Z 911.411,A -85,B 0,C 180,E1 14633.091,E2 14633.091} C_VEL
LIN {X 0,Y 334.705,Z 929.996,A -85,B 0,C 180,E1 14634.364,E2 14634.364} C_VEL
LIN {X 0,Y 330.302,Z 963.833,A -85,B 0,C 180,E1 14636.347,E2 14636.347} C_VEL
LIN {X 0,Y 325.037,Z 995.165,A -85,B 0,C 180,E1 14639.347,E2 14639.347} C_VEL
LIN {X 0,Y 319.673,Z 1022.878,A -85,B 0,C 180,E1 14643.261,E2 14643.261} C_VEL
LIN {X 0,Y 315.101,Z 1046.978,A -85,B 0,C 180,E1 14648.138,E2 14648.138} C_VEL
LIN {X 0,Y 312.322,Z 1066.335,A -85,B 0,C 180,E1 14653.815,E2 14653.815} C_VEL
LIN {X 0,Y 311.323,Z 1079.057,A -85,B 0,C 180,E1 14659.493,E2 14659.493} C_VEL
LIN {X 0,Y 311.455,Z 1085.724,A -85,B 0,C 180,E1 14664.422,E2 14664.422} C_VEL
LIN {X 0,Y 311.683,Z 1088.555,A -85,B 0,C 180,E1 14670.001,E2 14670.001} C_VEL
LIN {X 0,Y 311.406,Z 1086.445,A -85,B 0,C 180,E1 14675.581,E2 14675.581} C_VEL
LIN {X 0,Y 311.242,Z 1078.411,A -85,B 0,C 180,E1 14681.797,E2 14681.797} C_VEL
LIN {X 0,Y 312.845,Z 1064.413,A -85,B 0,C 180,E1 14687.972,E2 14687.972} C_VEL
LIN {X 0,Y 316.674,Z 1045.118,A -85,B 0,C 180,E1 14693.606,E2 14693.606} C_VEL
LIN {X 0,Y 322.259,Z 1021.524,A -85,B 0,C 180,E1 14698.406,E2 14698.406} C_VEL
LIN {X 0,Y 328.827,Z 993.713,A -85,B 0,C 180,E1 14702.363,E2 14702.363} C_VEL
LIN {X 0,Y 335.318,Z 962.358,A -85,B 0,C 180,E1 14705.348,E2 14705.348} C_VEL
LIN {X 0,Y 337.841,Z 947.539,A -85,B 0,C 180,E1 14706.344,E2 14706.344} C_VEL
LIN {X 0,Y 336.353,Z 937.373,A -85,B 0,C 180,E1 14707.281,E2 14707.281} C_VEL
LIN {X 0,Y 332.834,Z 927.61,A -85,B 0,C 180,E1 14708.362,E2 14708.362} C_VEL
LIN {X 0,Y 323.804,Z 901.802,A -85,B 0,C 180,E1 14710.91,E2 14710.91} C_VEL
LIN {X 0,Y 308.244,Z 872.838,A -85,B 0,C 180,E1 14714.524,E2 14714.524} C_VEL
LIN {X 0,Y 299.795,Z 858.394,A -85,B 0,C 180,E1 14716.726,E2 14716.726} C_VEL
LIN {X 0,Y 299.7,Z 857.28,A -85,B 0,C 180,E1 14716.958,E2 14716.958} C_VEL
LIN {X 0,Y 299.744,Z 857.28,A -85,B 0,C 180,E1 14723.922,E2 14723.922} C_VEL
LIN {X 0,Y 300.101,Z 857.28,A -85,B 0,C 180,E1 14732.966,E2 14732.966} C_VEL
LIN {X 0,Y 300.41,Z 857.28,A -85,B 0,C 180,E1 14739.311,E2 14739.311} C_VEL
LIN {X 0,Y 300.656,Z 857.28,A -85,B 0,C 180,E1 14745.385,E2 14745.385} C_VEL
LIN {X 0,Y 301.396,Z 857.28,A -85,B 0,C 180,E1 14754.199,E2 14754.199} C_VEL
LIN {X 0,Y 301.901,Z 857.28,A -85,B 0,C 180,E1 14759.963,E2 14759.963} C_VEL
LIN {X 0,Y 301.418,Z 857.28,A -85,B 0,C 180,E1 14765.726,E2 14765.726} C_VEL
LIN {X 0,Y 300.801,Z 857.28,A -85,B 0,C 180,E1 14774.532,E2 14774.532} C_VEL
LIN {X 0,Y 300.424,Z 857.28,A -85,B 0,C 180,E1 14780.609,E2 14780.609} C_VEL
LIN {X 0,Y 300.073,Z 857.28,A -85,B 0,C 180,E1 14786.954,E2 14786.954} C_VEL
LIN {X 0,Y 299.781,Z 857.356,A -85,B 0,C 180,E1 14794.294,E2 14794.294} C_VEL
LIN {X 0,Y 302.293,Z 863.006,A -85,B 0,C 180,E1 14795.079,E2 14795.079} C_VEL
LIN {X 0,Y 314.607,Z 887.238,A -85,B 0,C 180,E1 14799.152,E2 14799.152} C_VEL
LIN {X 0,Y 322.616,Z 911.142,A -85,B 0,C 180,E1 14803.038,E2 14803.038} C_VEL
LIN {X 0,Y 325.795,Z 932.581,A -85,B 0,C 180,E1 14806.696,E2 14806.696} C_VEL
LIN {X 0,Y 319.632,Z 955.55,A -85,B 0,C 180,E1 14810.565,E2 14810.565} C_VEL
LIN {X 0,Y 313.782,Z 973.691,A -85,B 0,C 180,E1 14815.189,E2 14815.189} C_VEL
LIN {X 0,Y 309.012,Z 987.012,A -85,B 0,C 180,E1 14820.66,E2 14820.66} C_VEL
LIN {X 0,Y 305.971,Z 994.562,A -85,B 0,C 180,E1 14826.678,E2 14826.678} C_VEL
LIN {X 0,Y 304.648,Z 996.055,A -85,B 0,C 180,E1 14832.65,E2 14832.65} C_VEL
LIN {X 0,Y 305.186,Z 991.88,A -85,B 0,C 180,E1 14838.553,E2 14838.553} C_VEL
LIN {X 0,Y 307.305,Z 981.803,A -85,B 0,C 180,E1 14844.344,E2 14844.344} C_VEL
LIN {X 0,Y 310.554,Z 966.423,A -85,B 0,C 180,E1 14849.524,E2 14849.524} C_VEL
LIN {X 0,Y 314.499,Z 947.253,A -85,B 0,C 180,E1 14853.795,E2 14853.795} C_VEL
LIN {X 0,Y 318.856,Z 922.634,A -85,B 0,C 180,E1 14857.502,E2 14857.502} C_VEL
LIN {X 0,Y 314.652,Z 898.137,A -85,B 0,C 180,E1 14860.747,E2 14860.747} C_VEL
LIN {X 0,Y 306.073,Z 870.836,A -85,B 0,C 180,E1 14863.732,E2 14863.732} C_VEL
LIN {X 0,Y 300.742,Z 857.28,A -85,B 0,C 180,E1 14865.052,E2 14865.052} C_VEL
LIN {X 0,Y 300.367,Z 857.28,A -85,B 0,C 180,E1 14870.661,E2 14870.661} C_VEL
LIN {X 0,Y 299.993,Z 857.28,A -85,B 0,C 180,E1 14877.015,E2 14877.015} C_VEL
LIN {X 0,Y 299.695,Z 857.28,A -85,B 0,C 180,E1 14883.76,E2 14883.76} C_VEL
LIN {X 0,Y 299.847,Z 857.28,A -85,B 0,C 180,E1 14890.315,E2 14890.315} C_VEL
LIN {X 0,Y 308.717,Z 888.268,A -85,B 0,C 180,E1 14892.403,E2 14892.403} C_VEL
LIN {X 0,Y 314.049,Z 914.43,A -85,B 0,C 180,E1 14894.987,E2 14894.987} C_VEL
LIN {X 0,Y 311.641,Z 939.583,A -85,B 0,C 180,E1 14898.092,E2 14898.092} C_VEL
LIN {X 0,Y 308.752,Z 961.869,A -85,B 0,C 180,E1 14902.172,E2 14902.172} C_VEL
LIN {X 0,Y 306.611,Z 978.552,A -85,B 0,C 180,E1 14906.779,E2 14906.779} C_VEL
LIN {X 0,Y 305.193,Z 990.251,A -85,B 0,C 180,E1 14911.937,E2 14911.937} C_VEL
LIN {X 0,Y 304.715,Z 995.824,A -85,B 0,C 180,E1 14916.628,E2 14916.628} C_VEL
LIN {X 0,Y 305.117,Z 997.153,A -85,B 0,C 180,E1 14920.53,E2 14920.53} C_VEL
LIN {X 0,Y 306.752,Z 994.22,A -85,B 0,C 180,E1 14925.756,E2 14925.756} C_VEL
LIN {X 0,Y 309.547,Z 985.517,A -85,B 0,C 180,E1 14930.99,E2 14930.99} C_VEL
LIN {X 0,Y 313.18,Z 972.095,A -85,B 0,C 180,E1 14935.532,E2 14935.532} C_VEL
LIN {X 0,Y 317.644,Z 952.599,A -85,B 0,C 180,E1 14939.728,E2 14939.728} C_VEL
LIN {X 0,Y 321.9,Z 928.805,A -85,B 0,C 180,E1 14943.066,E2 14943.066} C_VEL
LIN {X 0,Y 322.244,Z 914.918,A -85,B 0,C 180,E1 14944.682,E2 14944.682} C_VEL
LIN {X 0,Y 317.668,Z 892.234,A -85,B 0,C 180,E1 14947.328,E2 14947.328} C_VEL
LIN {X 0,Y 306.917,Z 868.768,A -85,B 0,C 180,E1 14950.412,E2 14950.412} C_VEL
LIN {X 0,Y 301.065,Z 858.853,A -85,B 0,C 180,E1 14952.097,E2 14952.097} C_VEL
LIN {X 0,Y 300.863,Z 857.28,A -85,B 0,C 180,E1 14952.382,E2 14952.382} C_VEL
LIN {X 0,Y 300.596,Z 857.28,A -85,B 0,C 180,E1 14957.622,E2 14957.622} C_VEL
LIN {X 0,Y 300.143,Z 857.28,A -85,B 0,C 180,E1 14964.77,E2 14964.77} C_VEL
LIN {X 0,Y 299.83,Z 857.28,A -85,B 0,C 180,E1 14970.858,E2 14970.858} C_VEL
LIN {X 0,Y 299.711,Z 857.28,A -85,B 0,C 180,E1 14977.344,E2 14977.344} C_VEL
LIN {X 0,Y 299.632,Z 857.28,A -85,B 0,C 180,E1 14985.054,E2 14985.054} C_VEL
LIN {X 0,Y 299.802,Z 857.885,A -85,B 0,C 180,E1 14988.515,E2 14988.515} C_VEL
LIN {X 0,Y 320.875,Z 908.851,A -85,B 0,C 180,E1 14992.183,E2 14992.183} C_VEL
LIN {X 0,Y 327.451,Z 931.867,A -85,B 0,C 180,E1 14993.843,E2 14993.843} C_VEL
LIN {X 0,Y 322.769,Z 965.644,A -85,B 0,C 180,E1 14995.947,E2 14995.947} C_VEL
LIN {X 0,Y 317.409,Z 996.116,A -85,B 0,C 180,E1 14998.996,E2 14998.996} C_VEL
LIN {X 0,Y 311.767,Z 1023.906,A -85,B 0,C 180,E1 15003.113,E2 15003.113} C_VEL
LIN {X 0,Y 307.312,Z 1046.68,A -85,B 0,C 180,E1 15007.935,E2 15007.935} C_VEL
LIN {X 0,Y 304.531,Z 1064.82,A -85,B 0,C 180,E1 15013.39,E2 15013.39} C_VEL
LIN {X 0,Y 303.488,Z 1077.689,A -85,B 0,C 180,E1 15019.218,E2 15019.218} C_VEL
LIN {X 0,Y 303.626,Z 1084.456,A -85,B 0,C 180,E1 15024.277,E2 15024.277} C_VEL
LIN {X 0,Y 303.867,Z 1087.362,A -85,B 0,C 180,E1 15030.001,E2 15030.001} C_VEL
LIN {X 0,Y 303.552,Z 1085.298,A -85,B 0,C 180,E1 15035.726,E2 15035.726} C_VEL
LIN {X 0,Y 303.358,Z 1078.342,A -85,B 0,C 180,E1 15041.517,E2 15041.517} C_VEL
LIN {X 0,Y 304.935,Z 1064.623,A -85,B 0,C 180,E1 15047.971,E2 15047.971} C_VEL
LIN {X 0,Y 308.883,Z 1045.725,A -85,B 0,C 180,E1 15053.803,E2 15053.803} C_VEL
LIN {X 0,Y 314.641,Z 1022.638,A -85,B 0,C 180,E1 15058.765,E2 15058.765} C_VEL
LIN {X 0,Y 321.748,Z 994.327,A -85,B 0,C 180,E1 15062.965,E2 15062.965} C_VEL
LIN {X 0,Y 328.611,Z 962.854,A -85,B 0,C 180,E1 15066.063,E2 15066.063} C_VEL
LIN {X 0,Y 333.493,Z 930.418,A -85,B 0,C 180,E1 15068.1,E2 15068.1} C_VEL
LIN {X 0,Y 332.834,Z 927.61,A -85,B 0,C 180,E1 15068.362,E2 15068.362} C_VEL
LIN {X 0,Y 327.89,Z 917.903,A -85,B 0,C 180,E1 15069.629,E2 15069.629} C_VEL
LIN {X 0,Y 317.145,Z 903.31,A -85,B 0,C 180,E1 15071.93,E2 15071.93} C_VEL
LIN {X 0,Y 301.723,Z 874.731,A -85,B 0,C 180,E1 15075.753,E2 15075.753} C_VEL
LIN {X 0,Y 291.854,Z 858.264,A -85,B 0,C 180,E1 15078.518,E2 15078.518} C_VEL
LIN {X 0,Y 291.79,Z 857.28,A -85,B 0,C 180,E1 15078.59,E2 15078.59} C_VEL
LIN {X 0,Y 291.863,Z 857.28,A -85,B 0,C 180,E1 15086.103,E2 15086.103} C_VEL
